ABB RAPID module: ComBase_LU.sys

MODULE ComBase_LU(SYSMODULE,NOSTEPIN)
!**********************************************************************
!* Dieses Module definiert  generellen Ablauf / Kommunikation zur SPS *
!* This module defines the general process / communication with PLC   *
!*                                                                    *
!*                Variablen und Einstellungen fuer die SPS            *
!*                   Variables and settings for PLC                   *
!**********************************************************************
! TypID Nummer fuer alle Applikationen
RECORD TypId
  num TypId_num;
ENDRECORD
!Module Version Number
CONST string st_Version_ComBase:="10.3.6c Test ComBase_LU";
 !Update 13th Apr 2015

! Automatische Einstellung der Sprache / Auto Setting for the language
! Abfrage des FlexPendant / request the FlexPendant
! 1=English, 2=Deutsch, 3=???
PERS num n_Sp:=1;
!
! Merker fuer die Applikationen, wird mit PowerOn neu gelesen / Marker for the applications is read when PowerOn
PERS string st_Appl_Info{30,3}:=[["2","Gripp Ware     ","1 = Actuator, 2 = PP->PLC, 3 = Setup"],["24","INOS Best Fit  ","1 = , 2 = , 3 = Setup"],["","",""],["","",""],["","",""],
	["","",""],["","",""],["","",""],["","",""],["","",""],["","",""],["","",""],["","",""],
	["","",""],["","",""],["","",""],["","",""],["","",""],["","",""],["","",""],["","",""],
	["","",""],["","",""],["","",""],["","",""],["","",""],["","",""],["","",""],["","",""],["","",""]];
VAR string st_Appl_Name:="";
VAR string st_Appl_Key{3}:=["","",""];
PERS num n_ApplMax:=2;
PERS num n_Fk4ApplAktiv:=0;
PERS num n_Fk4ApplNum:=0;
PERS bool b_PwOnEnd:=TRUE;
PERS num n_SMPins{4}:=[5553,0,0,0];
TASK PERS bool b_Start_present{30}:=[TRUE,FALSE,TRUE,TRUE,TRUE,TRUE,TRUE,TRUE,TRUE,TRUE,TRUE,TRUE,TRUE,TRUE,TRUE,
								TRUE,TRUE,TRUE,TRUE,TRUE,TRUE,TRUE,TRUE,TRUE,TRUE,TRUE,TRUE,TRUE,TRUE,TRUE];
PERS bool b_ReStart_present{30}:=[TRUE,FALSE,TRUE,TRUE,TRUE,TRUE,TRUE,TRUE,TRUE,TRUE,TRUE,TRUE,TRUE,TRUE,TRUE,
								  TRUE,TRUE,TRUE,TRUE,TRUE,TRUE,TRUE,TRUE,TRUE,TRUE,TRUE,TRUE,TRUE,TRUE,TRUE];
PERS bool b_Stop_present{30}:=[TRUE,FALSE,TRUE,TRUE,TRUE,TRUE,TRUE,TRUE,TRUE,TRUE,TRUE,TRUE,TRUE,TRUE,TRUE,
							   TRUE,TRUE,TRUE,TRUE,TRUE,TRUE,TRUE,TRUE,TRUE,TRUE,TRUE,TRUE,TRUE,TRUE,TRUE];
PERS bool b_Reset_present{30}:=[TRUE,TRUE,TRUE,TRUE,TRUE,TRUE,TRUE,TRUE,TRUE,TRUE,TRUE,TRUE,TRUE,TRUE,TRUE,
								TRUE,TRUE,TRUE,TRUE,TRUE,TRUE,TRUE,TRUE,TRUE,TRUE,TRUE,TRUE,TRUE,TRUE,TRUE];
PERS bool b_StartUser_present:=TRUE;
PERS bool b_ReStartUser_present:=TRUE;
PERS bool b_StopUser_present:=TRUE;
PERS bool b_ResetUser_present:=TRUE;
PERS bool b_PPMoved:=FALSE;
VAR bool b_PPMoved_mem:=FALSE;

VAR num n_Appl_count;
VAR bool b_UserEv;
!
! Variablen zum Dialog / Varaiables for Dialog
VAR string st_UiHeader{3};
VAR string st_UiHeader_2{3};
VAR string st_UiMsgLines{5};
VAR string st_UiMsgLine1{3};
VAR string st_UiMsgLine2{3};
VAR string st_UiMsgLine3{3};
VAR string st_UiMsgLine4{3};
VAR string st_UiMsgLine5{3};
VAR listitem li_UiMsgList{5};
VAR string st_UiMsgButtons{5};
VAR string st_UiMsgButtons1{3};
VAR string st_UiMsgButtons2{3};
VAR string st_UiMsgButtons3{3};
VAR string st_UiMsgButtons4{3};
VAR string st_UiMsgButtons5{3};
VAR string st_Dummy{3};
VAR string st_Dummy2{3};
VAR btnres br_UiAnswer;
!----------------------------------------------------
!Predefined Const for TypID
!
CONST TypId Id_00:=[0];
CONST TypId Id_01:=[1];
CONST TypId Id_02:=[2];
CONST TypId Id_03:=[3];
CONST TypId Id_04:=[4];
CONST TypId Id_05:=[5];
CONST TypId Id_06:=[6];
CONST TypId Id_07:=[7];
CONST TypId Id_08:=[8];
CONST TypId Id_09:=[9];
CONST TypId Id_10:=[10];
CONST TypId Id_11:=[11];
CONST TypId Id_12:=[12];
CONST TypId Id_13:=[13];
CONST TypId Id_14:=[14];
CONST TypId Id_15:=[15];
!----------------------------------------------------
! Variablen und Einstellungen der MsgBox die von den Appl gemeinsam genutzt werden /
! Variables and settings of the MsgBox that are shared by all Applications
VAR string st_MsgBoxHeader{3};
VAR string st_MsgBoxLine3{3};
VAR string st_MsgBoxLine4{3};
VAR string st_MsgBoxLine5{3};
VAR string st_MsgBoxElogLine4;
VAR string st_MsgBoxbutton1{3};
VAR string st_MsgBoxbutton2{3};
VAR string st_MsgBoxbutton3{3};
VAR string st_MsgBoxbutton4{3};
VAR string st_MsgBoxbutton5{3};
VAR string st_MsgBoxSignal;
VAR string st_MsgBoxSignalValue;
VAR string st_MsgBoxGeraeteName{3};
VAR num n_MsgBoxApplError;
VAR num n_MsgBoxPLC_Error;
VAR num n_MsgBoxGeraeteNr;
VAR num n_MsgBoxAnswer;
VAR num n_Step;
!----------------------------------------------------
! Variablen und Einstellungen der MsgBoxEventStart die von den Appl gemeinsam genutzt werden /
! Variables and settings of the MsgBoxEventStart that are shared by all Applications
VAR string st_MsgBoxEvHeader{3};
VAR string st_MsgBoxEvLine3{3};
VAR string st_MsgBoxEvLine4{3};
VAR string st_MsgBoxEvLine5{3};
VAR string st_MsgBoxEvElogLine4;
VAR string st_MsgBoxEvbutton1{3};
VAR string st_MsgBoxEvbutton2{3};
VAR string st_MsgBoxEvbutton3{3};
VAR string st_MsgBoxEvbutton4{3};
VAR string st_MsgBoxEVbutton5{3};
VAR string st_MsgBoxEvSignal;
VAR string st_MsgBoxEvSignalValue;
VAR string st_MsgBoxEvGeraeteName{3};
VAR num n_MsgBoxEvApplError;
VAR num n_MsgBoxEvPLC_Error;
VAR num n_MsgBoxEvGeraeteNr;
VAR num n_MsgBoxEvAnswer;
VAR num n_StepEv;
!----------------------------------------------------
! Kalibrierposition jpCalibA1_A6 Achsen1-6 auf 0 Grad / Calibration position
CONST jointtarget jpCalibA1_A6:=[ [ 0, 0, 0, 0, 0, 0],[0, 0, 0, 0, 0, 0]];
PERS jointtarget jpTemp:=[ [ 92.8961, 38.0687, 0, 0, 2, 1.67904E-07],[9E+09, 9E+09, 9E+09, 9E+09, 9E+09, 9E+09]];
!
VAR num n_HomeSelect;
VAR num n_PGNNumber;
PERS num n_PGNNumber_Mem:=1;!Last Program number memory

VAR num n_Temp;
VAR bool b_Temp;
VAR num n_JobFinNum;
VAR num n_JobReqNum;
VAR bool b_JobF_w;
VAR bool b_JobR_w;


!----------------------------------------------------
! Tool fuer Position jpSM1SyncSwitch / Tool information for jpSM1SyncSwitchpos position
TASK PERS tooldata t_SMSync:= [TRUE, [[0.04, -0.03, 66.92], [0.991445, 0, 0, 0.130526]],[26.5, [-58.6, 41.7, -18.4],[1, 0, 0, 0], 0, 0, 0.141]];
!
!**********************************************************
!Copy SM Files to HOME directory                         *
!**********************************************************
CONST string stSMCalInternal:="INTERNAL:/OPTIONS/PSC/psc_calib_";
CONST string stSMCalHome:="HOME:/SafetyBCK/psc_calib_";
CONST string stSMInternal:="INTERNAL:/OPTIONS/PSC/psc_user_";
CONST string stSMHome:="HOME:/SafetyBCK/psc_user_";
CONST string stSMBck:="/hd0a/BACKUP/";
CONST string stSMBckFile:="/HOME/SafetyBCK/psc_user_";
CONST string stSMBckCal:="/HOME/SafetyBCK/psc_calib_";

VAR string stCon_Int_Dir;  !Controller internal directory
VAR string stCon_Home_Dir; !Controller internal Home directory
VAR string sthd0a_Home_Dir;!Flash card internal Home directory

! Filesize of an empty SM user_config
CONST num nSMFilesize:=230;
!----------------------------------------------------
! Home Var
TASK PERS tooldata t_Home:= [TRUE, [[26.5774, 98.0613, 502.695], [0.608761, 0, 0, -0.793353]],[311.4, [-15.6, -0.4, 261.4],[1, 0, 0, 0], 130.469, 118.237, 123.004]];
TASK PERS wobjdata wobj_home:=[FALSE, TRUE, "", [[603,2050.01,-515], [0,0,0,1]], [[0,0,0], [1,0,0,0]]];
VAR speeddata sp_SpeedHome;
VAR listitem listHome{5};
!----------------------------------------------------
! Bezeichner fuer die Home, bleibt einsprachig / Identifier for the home, remains monolingual
CONST listitem listHomeConst{5} := [ ["","Home 1 "], ["","Home 2 "],["","Home 3 "],["","Home 4 "] ,["","Home 5 "]  ];
!----------------------------------------------------
! Home Posabweichung Fein 2 Grad fuer Weltzone Home Ueberwachung / Home position in position tolerance
CONST jointtarget delta_HomePosFine := [ [ 2, 2, 2, 2, 2, 2],[5, 5, 5, 5, 5, 5]];
!----------------------------------------------------
! Volumen-Daten Weltzone Home Ueberwachung / Volume of data world-zone Home Surveillance
VAR shapedata sh_HomePos1;
VAR shapedata sh_HomePos2;
VAR shapedata sh_HomePos3;
VAR shapedata sh_HomePos4;
VAR shapedata sh_HomePos5;
!----------------------------------------------------
! Weltzonen Home Ueberwachung / World Home Surveillance Zones
VAR wzstationary wz_HomePos1:=[0];
VAR wzstationary wz_HomePos2:=[0];
VAR wzstationary wz_HomePos3:=[0];
VAR wzstationary wz_HomePos4:=[0];
VAR wzstationary wz_HomePos5:=[0];
!----------------------------------------------------
! Kugel durchmesser Weltzonen Ueberwachung / Ball diameter world zones Surveillance
CONST num n_Ball:=50;
!----------------------------------------------------
! Merker fuer Kolisionsueberwachung / Marker for Collision control
PERS bool b_CollZoneOccupied{63}:=[FALSE,FALSE,FALSE,FALSE,FALSE,FALSE,FALSE,FALSE,FALSE,FALSE,FALSE,FALSE,FALSE,FALSE,FALSE,FALSE,FALSE,FALSE,FALSE,FALSE,FALSE,FALSE,FALSE,FALSE,FALSE,FALSE,FALSE,FALSE,FALSE,FALSE,FALSE,FALSE,FALSE,FALSE,FALSE,FALSE,FALSE,FALSE,FALSE,FALSE,FALSE,FALSE,FALSE,FALSE,FALSE,FALSE,FALSE,FALSE,FALSE,FALSE,FALSE,FALSE,FALSE,FALSE,FALSE,FALSE,FALSE,FALSE,FALSE,FALSE,FALSE,FALSE,FALSE];
PERS num n_Coll{5}:=[2,0,0,0,0];
PERS num n_CollClZ:=1;
PERS bool b_CollClearAct:=FALSE;
!----------------------------------------------------
! Merker fuer PP wurde versetzt
VAR bool b_CheckPP;
!----------------------------------------------------
! Fehlerausgabe Status / Error Status
VAR bool b_OK;
VAR bool b_TimeOut;
!----------------------------------------------------
! Merker fuer Produktions loop / Marker for production loops
VAR bool b_AutoOff;
! Betriebsstundenzaehler / operating hours counters
VAR string st_op_cnt:="";
PERS num n_op_h_counter:=5881;
VAR string st_Abs;
!----------------------------------------------------
VAR Bool b_MainProg_Started ;!A main program as been started
PERS Bool b_PowerOn_exe_OK:=TRUE ;!Power on event has been executed
PERS Bool b_TbCom_Started:=TRUE ;!Background TB Com started
PERS bool b_Ignore_NoAppl_Chk:=FALSE ;!Ignore No APpplication check in StartCOM
PERS num n_ModeOP_Mem:=1 ;!Keyswitch mode operation memory
VAR Bool b_PathColDetectOn:=FALSE ;!Motor supervision on
VAR num n_ManSyncCMD:=0;! ManSyncPos Command
!----------------------------------------------------
!Variables to Check if this robot absolute accuracy compitable
PERS String st_RobotType:="ROB1_7600_2.55_500" ;!Robot type
PERS Bool b_Robot_ABS_Type ;!Robot is absolute accurate
VAR Bool b_ABS_Acc_Enable:=TRUE ;!Application ignore Absolute accuracy message
!----------------------------------------------------

!MsgBox di Break Control
PERS String st_MsgboxBrk_SignalName ;!Message box break Signal name to TB_Com
PERS String st_MsgboxBrk_ReturnName ;!Message box break Return Signal name from TB_Com
PERS Dnum dn_MsgboxBrk_ReqValue ;!Message box break required value to TB_Com
PERS Bool b_Invert_Control ;!Message box break Inverse Control Output to TB_Com

!Variables for monitoring Safety Gate and Manual teach mode keyswitch
PERS Bool b_SafetyGate_Was_Opened ;!Safety Gate was opened
PERS Bool b_ManMode_Was_Selected ;!Manual mode was selected
PERS Num n_SafetyGate_Req_Time;! Time the safety gate must be opened before timeout
PERS Num n_SafetyGate_Opened_Time;! Time the safety gate has been opened

!Variables for Log system
PERS String s_LOG_TX_Data ;!Message to be entered into log max 50 char
PERS String s_LOG_TX_Cat  ;!Message Category into log max 4 char

!Variables for Bit level Group Input and Output control
VAR num  n_LastGroupOutput:=0;
VAR num  n_LastGroupInput:=0;

!Robot number used identify the robot used for this task mainly used for Multimove
CONST Num n_RobotNr:=1;

!Memorise plc Error code
PERS Num n_PLC_ErrCode_Mem:=-4;
!----------------------------------------------------


!Variables for Indirect_WOBJ
PERS num n_DefWob_jDiff_Ges{3}:=[2.09808E-05,0.264905,0.433745];
PERS num n_DefWobj_Diff_Z{3}:=[2.09808E-05,-0.00128365,0.00133324];
PERS num n_DefWobj_Diff_Y{3}:=[0,0.264893,-0.417847];
PERS num n_DefWobj_Diff_X{3}:=[0,-0.0022583,-0.116348];
PERS wobjdata wobj_DefWobj_car0:=[FALSE,TRUE,"",[[-1.55826,939.221,447.268],[0.707962,0.0617476,0.0581078,-0.701142]],[[0,0,0],[1,0,0,0]]];
PERS tooldata t_DefWobj_Act_tool:=[TRUE,[[0,0,0],[1,0,0,0]],[0.001,[0,0,0.001],[1,0,0,0],0,0,0]];
PERS wobjdata wobj_DefWobj_ACT_wobj:=[FALSE,TRUE,"",[[0,0,0],[1,0,0,0]],[[0,0,0],[1,0,0,0]]];
PERS string s_DefWobj_Tool_Name:="tool0";
PERS string s_DefWobj_Wobj_Name:="wobj0";
PERS num n_DefWobj_px:=2734.52;
PERS num n_DefWobj_py:=-250;
PERS num n_DefWobj_pz:=40.459;
PERS robtarget rt_DefWobj_user_p{3}:=[[[271.15,-1260.46,24.4443],[0.539391,-0.00995541,0.0179942,0.841804],[-1,-1,0,1],[9E+09,9E+09,9E+09,9E+09,9E+09,9E+09]],[[275.724,-1760.69,26.8719],[0.539275,-0.00995293,0.0180075,0.841877],[-1,-1,0,1],[9E+09,9E+09,9E+09,9E+09,9E+09,9E+09]],[[-224.132,-1764.6,23.8962],[0.539218,-0.00994843,0.0180428,0.841914],[-2,-2,0,1],[9E+09,9E+09,9E+09,9E+09,9E+09,9E+09]]];
PERS robtarget rt_DefWobj_mess_p{3}:=[[[2242.11,250,-46.365],[1,0,0,0],[-1,-1,-1,0],[9E+09,9E+09,9E+09,9E+09,9E+09,9E+09]],[[2734.52,250,40.459],[1,0,0,0],[-1,-1,-1,0],[9E+09,9E+09,9E+09,9E+09,9E+09,9E+09]],[[2734.52,-250,40.459],[1,0,0,0],[-1,-1,-1,0],[9E+09,9E+09,9E+09,9E+09,9E+09,9E+09]]];


!----------------------------------------------------

PROC InitAutoMode()
!******************************************************
!*                                                    *
!* Prozedur fuer das Starten des Roboters in Automatik*
!*   Procedure for starting the robot in automatic!   *
!*                                                    *
!******************************************************
!
! Bewegungsueberwachung einschalten / Activate motion supervision
MotionSup \On;

!Reset Msgbox signals
SetGO PLC_go_ErrCode, 0;
Reset PLC_do_MsgToPLC;
Reset PLC_do_ErrorToPLC;
Reset PLC_do_StopToPLC;
Reset VB_do_TaskBrake;
n_PLC_ErrCode_Mem:=-1;

! abfrage ob Betriebsart Hand / Check operation mode
WHILE OpMode()= OP_AUTO DO
	st_UiHeader:=["Com, Waiting for Robot in Teach Mode ","Com, Warte auf Hand-Betrieb","???"];
	st_UiMsgLine1:=["  Please switch the mode selection ","  Bitte Programm Main in der Betriebsart ","???"];
	st_UiMsgLine2:=["  to Teach/Manual Mode.","  Hand starten.","???"];
	UIMsgBox\Header:=st_UiHeader{n_Sp},st_UiMsgLine1{n_Sp}\MsgLine2:=st_UiMsgLine2{n_Sp}
	\Buttons:=btnOK\Icon:=iconWarning;
	!
	IF OpMode()= OP_AUTO Stop;
ENDWHILE

IF b_PowerOn_exe_OK=FALSE PowerOnCom ;

! Abfrage ob die AbsAcc ein ist
ReadCfgData "/MOC/ROBOT/ROB_1","use_robot_calib",st_Abs;

IF st_Abs="r1_uncalib" AND b_Robot_ABS_Type THEN
	st_UiHeader:=["Com, No Absolute Accuracy","Com, Keine Absolutgenauigkeit","???"];
	st_UiMsgLine1:=["Warning! The robot absolute accuracy is turned Off.","Achtung bei diesem Roboter ist die Absolutgenauigkeit = Off","???"];
	st_UiMsgLine2:=["Absolute accuracy must be enabled","Ohne aktive Absolutgenauigkeit ist es nicht erlaubt","???"];
	st_UiMsgLine3:=["and without it, there is a high risk ","den Roboter zu programmieren oder Programme abzufahren,","???"];
	st_UiMsgLine4:=["of a collision.","es besteht Kollisionsgefahr!","???"];
	st_UiMsgLine5:=["Please ensure it is enabled!","Bitte schalten Sie die Absolutgenauigkeit wieder ein!","???"];
    st_UiMsgButtons5:=["Ignore","ignorieren","???"];
    st_UiMsgButtons:=["","","","",st_UiMsgButtons5{n_Sp}];
    st_UiMsgLines:=[st_UiMsgLine1{n_Sp},st_UiMsgLine2{n_Sp},st_UiMsgLine3{n_Sp},st_UiMsgLine4{n_Sp},st_UiMsgLine5{n_Sp}];
    br_UiAnswer:=UIMessageBox (\Header:=st_UiHeader{n_Sp}\MsgArray:=st_UiMsgLines\BtnArray:=st_UiMsgButtons\Icon:=iconError);
ENDIF

! Abfrage ob der Roboter synchron ist / check because synced Robot
IF DOutput(SM1_do_Synced) = 0 THEN
	br_UiAnswer:=0;
	st_UiHeader:=["Com, SafeMove not Synchronised!","Com, SafeMove nicht synchron!","???"];
	st_UiMsgLine1:=["Warning! SafeMove(safety control) is not activated","Achtung, SafeMove(Sicherheitssteuerung) ist nicht aktiv!","???"];
	st_UiMsgLine2:=["Automatic operation without *SoftSync* is not possible!","Automatikbetrieb ist mit der Option *SoftSync* nicht moeglich!","???"];
	st_UiMsgLine3:=["Please synchronise the robot (SafeMove).","Bitte den Roboter (SafeMove) erst manuell synchronisieren lassen.","???"];
	st_UiMsgLine4:=["","","???"];
	st_UiMsgLine5:=["Press> Ignore to continue to operate without SoftSync.","Mit ignorieren geht es im Ablauf (ohne SoftSync) weiter.","???"];
	st_UiMsgButtons5:=["Ignore","ignorieren","???"];
	st_UiMsgButtons:=["","","","",st_UiMsgButtons5{n_Sp}];
	st_UiMsgLines:=[st_UiMsgLine1{n_Sp},st_UiMsgLine2{n_Sp},st_UiMsgLine3{n_Sp},st_UiMsgLine4{n_Sp},st_UiMsgLine5{n_Sp}];
	!
	br_UiAnswer:=UIMessageBox (\Header:=st_UiHeader{n_Sp}
	\MsgArray:=st_UiMsgLines\BtnArray:=st_UiMsgButtons\Icon:=iconWarning);
ENDIF

! Simulierte Signale Abfragen
IF DOutput(VB_do_Simulated_IO)= 1 AND RobOS() = TRUE  THEN
	WHILE DOutput(VB_do_Simulated_IO)= 1 DO
 		st_UiHeader:=["Com, Caution simulated signals!","Com, Achtung Simulierte Signale!","???"];
 		st_UiMsgLine1:=["There are some signals that are simulated which is not allowed in ","Das Simulieren von Signalen ist im Automatik nicht erlaubt!","???"];
 		st_UiMsgLine2:=["automatic mode!  To continue please","Um fortzufahren bitte die Simulation aller","???"];
 		st_UiMsgLine3:=["select the I/O menu then turn off the simulation/s.","Signale im Ein-Ausgangs Fenster ausschalten.","???"];
 		UIMsgBox\Header:=st_UiHeader{n_Sp},st_UiMsgLine1{n_Sp}\MsgLine2:=st_UiMsgLine2{n_Sp}\MsgLine3:=st_UiMsgLine3{n_Sp}
 						\Buttons:=btnOk\Icon:=iconWarning;
		!
		IF DOutput(VB_do_Simulated_IO)= 1 Stop;
	ENDWHILE
ENDIF

!Jog supervision enable
WriteCfgData "/MOC/MOTION_SUP/rob1","jog_col_detect_on", TRUE;

!Check motor supervision enabled
ReadCfgData "/MOC/MOTION_SUP/rob1","path_col_detect_on",b_PathColDetectOn;

IF b_PathColDetectOn=FALSE THEN
	st_UiHeader:=["Com, Motor Supervision","Com, Motor Ueberwachung","???"];
	st_UiMsgLine1:=["The robot path supervision is","Die Roboter Pfad Ueberwachung ist","???"];
	st_UiMsgLine2:=["turned off and should be turned on.","ausgeschalten und solle angeschalten sein.","???"];
	st_UiMsgLine3:=["","","???"];
	st_UiMsgLine4:=["","","???"];
	st_UiMsgLine5:=["Please select option.","Option waehlen bitte.","???"];
    st_UiMsgButtons4:=["Turn On","anschalten","???"];
    st_UiMsgButtons5:=["Ignore","ignorieren","???"];
    st_UiMsgButtons:=["","","",st_UiMsgButtons4{n_Sp},st_UiMsgButtons5{n_Sp}];
    st_UiMsgLines:=[st_UiMsgLine1{n_Sp},st_UiMsgLine2{n_Sp},st_UiMsgLine3{n_Sp},st_UiMsgLine4{n_Sp},st_UiMsgLine5{n_Sp}];
    br_UiAnswer:=UIMessageBox (\Header:=st_UiHeader{n_Sp}\MsgArray:=st_UiMsgLines\BtnArray:=st_UiMsgButtons\Icon:=iconWarning);

    IF br_UiAnswer=4 WriteCfgData "/MOC/MOTION_SUP/rob1","path_col_detect_on", TRUE;
ENDIF

! meldet an PLC das Programmzeiger im Main ist / Inform PLC main program is selected
b_CheckPP:=TRUE;
Set SYS_do_MainStarted;
VelSet 100,5000;

! zum anfahren der Homeposition
! abfrage ob mehr als eine HomePos / Check number of homes configured
FOR i FROM 1 TO 5 DO
  IF b_HomeInUse{i}=TRUE Incr n_Temp;
ENDFOR

! auslesen der Beschreibung der benutzten Home / Read the home descriptions
IF n_Temp>1 THEN
 	Abfrg2:
	FOR i FROM 1 TO 5 DO
		IF b_HomeInUse{i} THEN
			! vorgabe der Home von der SPS / specification of the Home of the PLC
			IF b_PLCNeedHome(i)= TRUE THEN
				st_UiMsgLine1:=["PLC> ","SPS> ","???"];
				listHome{i}.text:=st_UiMsgLine1{n_Sp};
			ELSE
				listHome{i}.text:="        ";
			ENDIF
			listHome{i}.text:=listHome{i}.text+listHomeConst{i}.text+st_Home_label{i};
		ELSE
			listHome{i}.text:="";
		ENDIF
	ENDFOR

	! Anzeigen der HomePos / Generate Home positions message
  	st_UiHeader:=["Com, The Robot is ","Com, Der Roboter steht auf ","???"];

	IF n_RobInHomeDO()> 0 THEN
    	st_UiHeader_2:=["at Home number "+ValToStr(n_RobInHomeDO()),"Home "+ValToStr(n_RobInHomeDO()),"???"+ValToStr(n_RobInHomeDO())];
	ELSE
    	st_UiHeader_2:=["not in any Home.","keiner Home.","???"];
	ENDIF

	st_UiMsgButtons1:=["Refresh Display","Ansicht aktualisieren","???"];
	st_UiMsgButtons4:=["Ok","Ok","???"];
	st_UiMsgButtons5:=["Abort","Abbruch","???"];
	st_UiMsgButtons:=[st_UiMsgButtons1{n_Sp},"","",st_UiMsgButtons4{n_Sp},""];

	n_HomeSelect := UIListView(\Result:=br_UiAnswer\Header:=st_UiHeader{n_Sp}+st_UiHeader_2{n_Sp},listHome
      \BtnArray:=st_UiMsgButtons\Icon:=iconInfo\DefaultIndex:=n_RobInHomeDO());

	IF br_UiAnswer = 1 GOTO Abfrg2;
	IF br_UiAnswer = 5 THEN
  	TPErase;
  	TPShow TP_LATEST;
  	EXIT ;
   ENDIF
ELSE !n_temp>1
	! es gibt nur eine Home / There is only one Home
	n_HomeSelect:=1;
ENDIF !n_temp>1

!----------------------------------------------------
! Ueberprueft ob die Homeposition programmiert wurde / Checks whether the home position has been programmed
br_UiAnswer:=0;
b_Temp:=FALSE;
IF n_HomeSelect=1 AND jpHome1.robax <> jpCalibA1_A6.robax AND b_HomeAkt{n_HomeSelect}=TRUE b_Temp:=TRUE;
IF n_HomeSelect=2 AND jpHome2.robax <> jpCalibA1_A6.robax AND b_HomeAkt{n_HomeSelect}=TRUE b_Temp:=TRUE;
IF n_HomeSelect=3 AND jpHome3.robax <> jpCalibA1_A6.robax AND b_HomeAkt{n_HomeSelect}=TRUE b_Temp:=TRUE;
IF n_HomeSelect=4 AND jpHome4.robax <> jpCalibA1_A6.robax AND b_HomeAkt{n_HomeSelect}=TRUE b_Temp:=TRUE;
IF n_HomeSelect=5 AND jpHome5.robax <> jpCalibA1_A6.robax AND b_HomeAkt{n_HomeSelect}=TRUE b_Temp:=TRUE;

IF b_Temp=FALSE THEN
	st_UiHeader:=["Com, Home Configuration Error","Com, Fehlerhafte Home_","Com,???"];
	IF b_HomeAkt{n_HomeSelect}=FALSE THEN
		st_UiMsgLine1:=["The Home position selected has not been activated","Die ausgewaehlte Home ist nicht aktiv","???"];
		st_UiMsgLine2:=["therefore, the Home output will not be sent to the PLC.","der Ausgang wird nicht zur SPS gesetzt.","???"];
		st_UiMsgLine3:=["Please select 'HomeSetup' to configure.","Bitte ueber das HomeSetup die Home aktivieren.","???"];
	ELSE
		st_UiMsgLine1:=["The Home position selected either not programmed","Die ausgewaehlte Home ist nicht programmiert","???"];
		st_UiMsgLine2:=["or the robot is in the calibration position!","oder entspricht der Nullstellung!","???"];
		st_UiMsgLine3:=["Please select 'Setup' to configure.","Bitte die Position ueber das HomeSetup anpassen.","???"];
	ENDIF

	st_UiMsgButtons3:=["Home Setup","Home Setup","???"];
	st_UiMsgButtons5:=["Abort","Abbruch","???"];
	st_UiMsgButtons:=["","",st_UiMsgButtons3{n_Sp},"",st_UiMsgButtons5{n_Sp}];
	st_UiMsgLines:=[st_UiMsgLine1{n_Sp},st_UiMsgLine2{n_Sp},st_UiMsgLine3{n_Sp},"",""];

	br_UiAnswer:=UIMessageBox (\Header:=st_UiHeader{n_Sp}+ValToStr(n_HomeSelect)
		\MsgArray:=st_UiMsgLines\BtnArray:=st_UiMsgButtons\Icon:=iconWarning);

	IF br_UiAnswer = 5 THEN
		TPErase;
		TPShow TP_LATEST;
		EXIT;
	ENDIF

	IF br_UiAnswer = 3 Homesetup;
	EXIT;
ENDIF

! Abfrage wegen Tool 0 / check because of tool zero
IF CTool()=tool0 THEN
  	br_UiAnswer:=0;
  	st_UiHeader:=["Com, Tool Load check","Com, Tool Ueberpruefung","???"];
  	st_UiMsgLine1:=["Attention!! the active tool is tool0.","Achtung das aktive Tool ist - tool0 - !!! ","???"];
  	st_UiMsgLine2:=["The robot cannot move with tool0 because","Der Roboter kann vermutlicht wegen falschen  ","???"];
  	st_UiMsgLine3:=["it has the incorrect payload configured.","Gewichtsdaten nicht bewegt werden, ","???"];
  	st_UiMsgLine4:=["Using the Jogging Window, please change to the","bitte waehle im Bewegen-Fenster das richtige Tool aus,","???"];
  	st_UiMsgLine5:=["correct tool then select 'Ok' button.","bevor es mit Ok weiter geht.","???"];
  	st_UiMsgButtons1:=["","","???"];
  	st_UiMsgButtons2:=["","","???"];
  	st_UiMsgButtons3:=["","","???"];
  	st_UiMsgButtons4:=["Ok","Ok","???"];
  	st_UiMsgButtons5:=["","","???"];
  	st_UiMsgButtons:=[st_UiMsgButtons1{n_Sp},st_UiMsgButtons2{n_Sp},st_UiMsgButtons3{n_Sp},st_UiMsgButtons4{n_Sp},st_UiMsgButtons5{n_Sp}];
  	st_UiMsgLines:=[st_UiMsgLine1{n_Sp},st_UiMsgLine2{n_Sp},st_UiMsgLine3{n_Sp},st_UiMsgLine4{n_Sp},st_UiMsgLine5{n_Sp}];
  	!
  	br_UiAnswer:=UIMessageBox (\Header:=st_UiHeader{n_Sp}
  	\MsgArray:=st_UiMsgLines\BtnArray:=st_UiMsgButtons\Icon:=iconWarning);
ENDIF

! Bestaetigung und Geschwindigkeitsauswahl / Confirmation and speed selection
sp_SpeedHome:=v100;
IF b_RobInHomeDO(n_HomeSelect)= FALSE THEN
  	br_UiAnswer:=0;
  	st_UiHeader:=["Com, Move Robot to Homepos ","Com, Bewege Roboter zur Home ","Com,???"];
  	st_UiMsgLine3:=["     Attention!","    Achtung!","???"];
  	st_UiMsgLine4:=["     The Robot will move -> ","    Roboter faehrt mit Ok -> ","???"];
  	st_UiMsgLine5:=["     directly to the Home ","    direkt zur Home ","???"];
  	st_UiMsgButtons1:=["Fast (v250)","SCHNELL (v250)","???"];
  	st_UiMsgButtons2:=["Slow (v100)","LANGSAM (v100)","???"];
  	st_UiMsgButtons3:=["","","???"];
  	st_UiMsgButtons4:=["Move Home","Ok","???"];
  	st_UiMsgButtons5:=["Abort","Abbruch","???"];
  	st_UiMsgButtons:=[st_UiMsgButtons1{n_Sp},st_UiMsgButtons2{n_Sp},st_UiMsgButtons3{n_Sp},st_UiMsgButtons4{n_Sp},""];
  	st_Dummy:=st_UiMsgButtons2;
  	Abfrg1:
  	st_UiMsgLines:=[" "," ",st_UiMsgLine3{n_Sp},st_UiMsgLine4{n_Sp}+st_Dummy{n_Sp},st_UiMsgLine5{n_Sp}+ValToStr(n_HomeSelect)];

  	br_UiAnswer:=UIMessageBox (\Header:=st_UiHeader{n_Sp}+ValToStr(n_HomeSelect)
  			\MsgArray:=st_UiMsgLines\BtnArray:=st_UiMsgButtons\Icon:=iconWarning);

	TEST br_UiAnswer
		CASE 1:
		! schnell/fAST
		st_Dummy:=st_UiMsgButtons1;
		sp_SpeedHome:=v200;
		GOTO Abfrg1;
	CASE 2:
		! langsam/sLOW
		st_Dummy:=st_UiMsgButtons2;
		sp_SpeedHome:=v100;
		GOTO Abfrg1;
	CASE 4:
		! OK/ok
	CASE 5:
		! Abbruch / Abort
		TPErase;
		TPShow TP_LATEST;
			EXIT;
	ENDTEST

	! Prozedur zum Initialisieren von Ein-, Ausgaengen, Variabelen fuer den User / Procedure to initialize inputs, outputs, variables for the user
	InitBeforHome n_HomeSelect;
	! Homefahrt
	t_Home := CTool();
	wobj_home := CWobj();

	TEST n_HomeSelect
	CASE 1:
		MoveAbsJ jpHome1\NoEOffs, sp_SpeedHome, fine, t_Home\WObj:=wobj_home;
	CASE 2:
		MoveAbsJ jpHome2\NoEOffs, sp_SpeedHome, fine, t_Home\WObj:=wobj_home;
	CASE 3:
		MoveAbsJ jpHome3\NoEOffs, sp_SpeedHome, fine, t_Home\WObj:=wobj_home;
	CASE 4:
		MoveAbsJ jpHome4\NoEOffs, sp_SpeedHome, fine, t_Home\WObj:=wobj_home;
	CASE 5:
		MoveAbsJ jpHome5\NoEOffs, sp_SpeedHome, fine, t_Home\WObj:=wobj_home;
	ENDTEST
ELSE !n_HomeSelect
	! Roboter steht schon auf Home x
	! Prozedur zum Initialisieren von Ein-, Ausgaengen, Variabelen fuer den User /
	! Robots already standing at home x
	! Procedure to initialize inputs, outputs, variables for the user
 	InitBeforHome n_HomeSelect;
ENDIF !n_HomeSelect

! check ob Home x Ausgang = 1
IF b_RobInHomeDO(n_HomeSelect)= FALSE THEN
  	br_UiAnswer:=0;
  	st_UiHeader:=["Com, Error Output SYS_do_Home_"+ValToStr(n_HomeSelect)+" = 0","Com, Fehler: Ausgang SYS_do_Home_"+ValToStr(n_HomeSelect)+" = 0","Com,???"];
  	st_UiMsgLine3:=[" Attention Output from Home "+ValToStr(n_HomeSelect)+" does not =1.","Achtung der Ausgang fuer die Home " +ValToStr(n_HomeSelect)+" wurde nicht gesetzt!","???"];
  	st_UiMsgLine4:=[" The HomePos is not valid therefore, the program will stop.","Die Grundstellung ist nicht gueltig, der Ablauf wird abgebrochen.","???"];
  	st_UiMsgLine5:=[" Please ReCheck the Home"+ValToStr(n_HomeSelect)+" using the HomeSetup option.","Bitte im HomeSetup die Grundstellung Home"+ValToStr(n_HomeSelect)+"  berichtigen. ","???"];
  	st_UiMsgButtons1:=["","","???"];
  	st_UiMsgButtons2:=["","","???"];
  	st_UiMsgButtons3:=["Home Setup","Home Setup","???"];
  	st_UiMsgButtons4:=["Ok","Ok","???"];
  	st_UiMsgButtons5:=["","","???"];
  	st_UiMsgButtons:=[st_UiMsgButtons1{n_Sp},st_UiMsgButtons2{n_Sp},st_UiMsgButtons3{n_Sp},st_UiMsgButtons4{n_Sp},st_UiMsgButtons5{n_Sp}];
  	st_UiMsgLines:=[" "," ",st_UiMsgLine3{n_Sp},st_UiMsgLine4{n_Sp},st_UiMsgLine5{n_Sp}];
  	!
  	br_UiAnswer:=UIMessageBox (\Header:=st_UiHeader{n_Sp}\MsgArray:=st_UiMsgLines\BtnArray:=st_UiMsgButtons\Icon:=iconError);
  	! Fehler /Error
    IF br_UiAnswer = 3 Homesetup;
  	TPErase;
  	TPShow TP_LATEST;
 	EXIT;
ENDIF

InitInHome n_HomeSelect;

! Prozedur zum Initialisieren von Ein-, Ausgaengen, Variabelen fuer den User /
! Procedure to initialize user inputs, outputs and variables
InitMain;
InitProduktion;

WHILE OpMode()<>OP_AUTO DO
	! Aufforderung fuer Automaikbetrieb
	br_UiAnswer:=0;
	st_UiHeader:=["Com, Automatic Mode","Com, Automatik Extern Betrieb","Com,???"];
	st_UiMsgLine2:=["Please turn the mode selection Switch ","Den Schluesselschalter auf Automatik stellen ","???"];
	st_UiMsgLine3:=["to the Automatic Mode External position.","um in die Betriebsart Automatik Extern ","???"];
	st_UiMsgLine4:=[" ","zu wechseln.","???"];
	st_UiMsgButtons5:=["Abort","Abbruch","???"];
	st_UiMsgButtons:=["","","","",""];
	st_UiMsgLines:=[" ",st_UiMsgLine2{n_Sp},st_UiMsgLine3{n_Sp},st_UiMsgLine4{n_Sp},""];

	br_UiAnswer:=UIMessageBox (\Header:=st_UiHeader{n_Sp}
		\MsgArray:=st_UiMsgLines\BtnArray:=st_UiMsgButtons\Icon:=iconInfo\DOBreak:=SYS_do_Auto);
	!
	IF br_UiAnswer = resCancel THEN
		TPErase;
		TPShow TP_LATEST;
		EXIT;
	ENDIF
ENDWHILE

! Schleife fuer den AutoEX Betrieb\Loop for the operational AutoEX
WHILE b_AutoOff=FALSE DO
	b_AutoOff:=FALSE;
	InitProduktion;
	! Betriebsstundenzaehler lesen / operating hours counters read
	st_op_cnt:=GetServiceInfo(ROB_ID \DutyTimeCnt);
	b_Temp:=StrToVal(st_op_cnt, n_op_h_counter);

	WHILE SYS_di_ProgNumValid=1 DO
		st_MsgBoxHeader:=["Com, Error Prog Number Valid ","Com, Fehler Signal Prognum. gueltig!","???"];
		st_MsgBoxLine4:=["The Error is in the PLC","Fehlerbehebung an der SPS","???"];
		st_MsgBoxbutton4:=["Ok","Ok","???"];
		st_MsgBoxSignal:="SYS_di_ProgNumValid";
		st_MsgBoxGeraeteName:=["PLC I/O","SPS E/A","???"];
		n_MsgBoxGeraeteNr:=0;
		st_MsgBoxSignalValue:="0";
		n_MsgBoxApplError:=3;
		n_MsgBoxPLC_Error:=33;
		st_MsgBoxElogLine4:="ComBase/InitAutoMode";
		MsgBox\diBreakSignal:=SYS_di_ErrReset\ErrorToPLC;
	ENDWHILE

	! Betriebsstundenzaehler setzen zur SPS/ operating hours counters set to PLC
	IF b_Temp = TRUE SetGO PLC_go_WeldPoint_Num, n_op_h_counter;
	! anfrage Prognum. / Send program number request
	Set SYS_do_ProgNumReq;

	IF RobOS()  THEN
		st_UiHeader:=["          Com, Program Number","Com, Warte auf gueltige Programmnummer...","Com,???"];
		st_UiMsgLine1:=["         ******************************************","        ******************************************","???"];
		st_UiMsgLine2:=["         *     Waiting for the Program Number     *","        *      Warten auf die Programmnummer     *","???"];
		st_UiMsgLine3:=["         *              from the PLC.         V3.6*","        *               von der SPS.         V3.6*","???"];
		st_UiMsgLine4:=["         ******************************************","        ******************************************","???"];
		! Meldung an SPS, warte auf programmnummer / Waiting PLC Number
		 Reset PLC_do_ErrorToPLC;
		SetGO PLC_go_ErrCode, 32;
		Set PLC_do_MsgToPLC;
  		UIMsgBox\Header:=st_UiHeader{n_Sp},st_UiMsgLine1{n_Sp}\MsgLine2:=st_UiMsgLine2{n_Sp}
				\MsgLine3:=st_UiMsgLine3{n_Sp}\MsgLine4:=st_UiMsgLine4{n_Sp}\Buttons:=btnNone\Icon:=iconInfo
				\DIBreak:=SYS_di_ProgNumValid;
		! zuweisung der Prognum / Allocation of program number
		n_PGNNumber:=GInput(SYS_gi_ProgNumber);
		SetGO PLC_go_ErrCode, 0;
 		Reset PLC_do_MsgToPLC;
 		Reset PLC_do_ErrorToPLC;
	ELSE
		! manuelle Prognr nur fuer RobotStudio / Manual PGNR robot studio
  		st_UiHeader:=[" VirtualProgram Number","Programmnummer Virtual","???"];
 		st_UiMsgLine1:=["Program Number?","Programmnummer? 1-63","???"];
		n_PGNNumber := UINumEntry(\Header:=st_UiHeader{n_Sp}\Message:=st_UiMsgLine1{n_Sp}\Icon:=iconInfo
		\InitValue:=1\MinValue:=1\MaxValue:=63\AsInteger);
	ENDIF
	! Abfrage ob die AbsAcc ein ist
	ReadCfgData "/MOC/ROBOT/ROB_1","use_robot_calib",st_Abs;

	IF st_Abs="r1_uncalib" AND b_Robot_ABS_Type THEN
		st_UiHeader:=["Com, AbsAcc error","Com, Fehler Absolutgenauigkeit","???"];
		st_UiMsgLine1:=["Warning! The robot absolute accuracy is turned Off.","Achtung bei diesem Roboter ist die AbsAcc = Off","???"];
		st_UiMsgLine2:=["Absolute accuracy must be enabled","Ohne aktive Absolutgenauigkeit ist es nicht erlaubt","???"];
		st_UiMsgLine3:=["and without it, there is a high risk","den Roboter zu programmieren oder Programme abzufahren","???"];
		st_UiMsgLine4:=["of a collision.","es besteht Kollisionsgefahr!","???"];
		st_UiMsgLine5:=["Please ensure it is enabled!","Bitte schalten Sie die Absolutgenauigkeit wieder ein!","???"];
		UIMsgBox\Header:=st_UiHeader{n_Sp}, st_UiMsgLine1{n_Sp}\MsgLine2:=st_UiMsgLine2{n_Sp}\MsgLine3:=st_UiMsgLine3{n_Sp}
						\MsgLine4:=st_UiMsgLine4{n_Sp}\MsgLine5:=st_UiMsgLine5{n_Sp}\Buttons:=btnOK\Icon:=iconWarning;
	ENDIF

	n_PGNNumber_Mem:=n_PGNNumber;

	Reset SYS_do_ProgNumReq;
	SetGO PLC_go_WeldPoint_Num,0;
	! aufruf des Programms / Call program number
	Set SYS_do_ApplRun;
	%"Program_"+NumToStr(n_PGNNumber,0)%;
	Reset SYS_do_ApplRun;
ENDWHILE

ERROR
!** Error Handler**
! Fehlerbehandlung von nicht vorhandenen ProgNr. / None existant program number
SkipWarn;
IF ERRNO = ERR_REFUNKPRC THEN
    st_MsgBoxHeader:=["Com, Incorrect Program Number Call ","Com, Falsche Programm Nr. von der SPS!","???"];
    st_Dummy:=["The Routine called Program_"+ValToStr (n_PGNNumber),"Keine Routine Program_"+ValToStr (n_PGNNumber),"???"];
    st_Dummy2:=["was requested but is not programmed!!","im System vorhanden !","???"];
    st_MsgBoxbutton4:=["OK","Ok","???"];
    n_MsgBoxApplError:=0;
    n_MsgBoxPLC_Error:=31;
    st_MsgBoxElogLine4:="ComBase/InitAutoMode";
    MsgBox\diBreakSignal:=SYS_di_ErrReset\Line1:=st_Dummy{n_Sp}\Line2:=st_Dummy2{n_Sp}\ErrorToPLC;
  	TRYNEXT;
ENDIF
SkipWarn;
IF ERRNO = ERR_TP_DOBREAK TRYNEXT;
IF ERRNO = ERR_TP_DIBREAK TRYNEXT;
ENDPROC !(InitAutoMode)

!*******************************************************************************

PROC InitMain()
!**********************
!* Procedure InitMain *
!*   Intialise Main   *
!**********************
! Prozedur zum Initialisieren von Ein-, Ausgaengen, Variabelen / Procedure to initialize inputs, outputs, variables
! Procedur wird 1x im Main aufgerufen / First procedure called from main
 VAR bool b_ComDummy:=FALSE;
 VAR num n_ComDummy:=0;
!
 Reset SYS_do_ProgNumReq;
 Reset SYS_do_ApplRun;
 SetGO PLC_go_ErrCode, 0;
 Reset PLC_do_MsgToPLC;
 Reset PLC_do_ErrorToPLC;
 Reset PLC_do_StopToPLC;
 Reset PLC_do_CollZoneClear;
 Reset PLC_do_CollZoneReq;
 SetGO PLC_go_CollZone, 0;

 CollSafetyInit;
 b_AutoOff:=FALSE;
 n_JobReqNum:=0;
 n_JobFinNum:=0;
 b_JobF_w:=FALSE;
 b_JobR_w:=FALSE;
 !
 Reset PLC_do_Job01_Ready;
 Reset PLC_do_Job02_Ready;
 Reset PLC_do_Job03_Ready;
 Reset PLC_do_Job04_Ready;
 Reset PLC_do_Job05_Ready;
 Reset PLC_do_Job06_Ready;
 Reset PLC_do_Job07_Ready;
 Reset PLC_do_Job08_Ready;
 Reset PLC_do_Job09_Ready;
 Reset PLC_do_Job10_Ready;
 Reset PLC_do_Job11_Ready;
 Reset PLC_do_Job12_Ready;
 Reset PLC_do_Job13_Ready;
 Reset PLC_do_Job14_Ready;
 Reset PLC_do_Job15_Ready;
 Reset PLC_do_Job16_Ready;
 Reset PLC_do_Job17_Ready;
 Reset PLC_do_Job18_Ready;
 Reset PLC_do_Job19_Ready;
 Reset PLC_do_Job20_Ready;
 Reset PLC_do_Job21_Ready;
 Reset PLC_do_Job22_Ready;
 Reset PLC_do_Job23_Ready;
 Reset PLC_do_Job24_Ready;
 Reset PLC_do_Job25_Ready;
 Reset PLC_do_Job26_Ready;
 Reset PLC_do_Job27_Ready;
 Reset PLC_do_Job28_Ready;
 Reset PLC_do_Job29_Ready;
 Reset PLC_do_Job30_Ready;
 Reset PLC_do_Job31_Ready;
 Reset PLC_do_Job32_Ready;
 !
 Reset PLC_do_Job01_Started;
 Reset PLC_do_Job02_Started;
 Reset PLC_do_Job03_Started;
 Reset PLC_do_Job04_Started;
 Reset PLC_do_Job05_Started;
 Reset PLC_do_Job06_Started;
 Reset PLC_do_Job07_Started;
 Reset PLC_do_Job08_Started;
 Reset PLC_do_Job09_Started;
 Reset PLC_do_Job10_Started;
 Reset PLC_do_Job11_Started;
 Reset PLC_do_Job12_Started;
 Reset PLC_do_Job13_Started;
 Reset PLC_do_Job14_Started;
 Reset PLC_do_Job15_Started;
 Reset PLC_do_Job16_Started;
 Reset PLC_do_Job17_Started;
 Reset PLC_do_Job18_Started;
 Reset PLC_do_Job19_Started;
 Reset PLC_do_Job20_Started;
 Reset PLC_do_Job21_Started;
 Reset PLC_do_Job22_Started;
 Reset PLC_do_Job23_Started;
 Reset PLC_do_Job24_Started;
 Reset PLC_do_Job25_Started;
 Reset PLC_do_Job26_Started;
 Reset PLC_do_Job27_Started;
 Reset PLC_do_Job28_Started;
 Reset PLC_do_Job29_Started;
 Reset PLC_do_Job30_Started;
 Reset PLC_do_Job31_Started;
 Reset PLC_do_Job32_Started;
 !
 Reset PLC_do_Typbit_01;
 Reset PLC_do_Typbit_02;
 Reset PLC_do_Typbit_03;
 Reset PLC_do_Typbit_04;
 Reset PLC_do_Typbit_05;
 Reset PLC_do_Typbit_06;
 Reset PLC_do_Typbit_07;
 Reset PLC_do_Typbit_08;
 Reset PLC_do_Typbit_09;
 Reset PLC_do_Typbit_10;
 Reset PLC_do_Typbit_11;
 Reset PLC_do_Typbit_12;
 Reset PLC_do_Typbit_13;
 Reset PLC_do_Typbit_14;
 Reset PLC_do_Typbit_15;
 Reset PLC_do_Typbit_16;
 Reset PLC_do_Typbit_17;
 Reset PLC_do_Typbit_18;
 Reset PLC_do_Typbit_19;
 Reset PLC_do_Typbit_20;
 Reset PLC_do_Typbit_21;
 Reset PLC_do_Typbit_22;
 Reset PLC_do_Typbit_23;
 Reset PLC_do_Typbit_24;
 Reset PLC_do_Typbit_25;
 Reset PLC_do_Typbit_26;
 Reset PLC_do_Typbit_27;
 Reset PLC_do_Typbit_28;
 Reset PLC_do_Typbit_29;
 Reset PLC_do_Typbit_30;
 Reset PLC_do_Typbit_31;
 Reset PLC_do_Typbit_32;

 Reset PLC_do_ServicePos;
 Reset PLC_do_Process_Complete;
 Reset PLC_do_WeldCount;

 !Set output as this robot does not use this output
 IF st_RobotType="ROB1_6620LX_1.90_150" Set SM1_do_Stopped;

 ! aufruf der einzelnen Init Appl / calling the individual Init Appl
 IF n_ApplMax >0 AND n_ApplMax< 31 THEN
   FOR I FROM 1 TO n_ApplMax DO
     IF st_Appl_Info{I,1}="" GOTO END_InitAppl;
     b_ComDummy:=StrToVal(st_Appl_Info{I,1},n_ComDummy);
     %"InitAppl"+NumToStr(n_ComDummy,0)%;
   ENDFOR
 ENDIF
 END_InitAppl:
 ERROR
 !** Error Handler**
 SkipWarn;
 IF ERRNO=ERR_REFUNKPRC TRYNEXT;
ENDPROC !(InitMain)

!*******************************************************************************

PROC JobRequest()
!*************************************************************
!* Befehl Jobanfrage an die SPS / Command Job request to PLC *
!* Trap-Routine                                              *
!*************************************************************
VAR signaldo PLC_JobStarted;
VAR string st_alias2;
CONST string st_C:="PLC_do_Job";
CONST string st_D:="_Started";
!
IF n_JobReqNum>0 THEN
	! Signalnamen erzeugen / signalname to procreate
	IF n_JobReqNum <10 THEN
		st_alias2 :=st_C+"0"+NumToStr(n_JobReqNum,0)+st_D;
	ELSE
		st_alias2 :=st_C+NumToStr(n_JobReqNum,0)+st_D;
	ENDIF
	AliasIO st_alias2, PLC_JobStarted;
	!
  	Set PLC_JobStarted;
ELSE
	! Fehler Jobnum = 0
	ErrWrite \W, "PLC, Trap JobRequest error", "JobNum = 0" ;
ENDIF
n_JobReqNum:=0;
b_JobR_w:=FALSE;
ENDPROC !(JobRequest)

!*******************************************************************************

PROC MoveJ_JobRequest (num Job,  robtarget ToPoint,  speeddata Speed,  zonedata Zone,  PERS tooldata Tool  \PERS wobjdata Wobj)
!*************************************************
!*   Command to call the  job request routine    *
!* synchronous from a joint type motion movement *
!*************************************************
VAR signaldi PLC_JobEnable;
VAR string st_alias;
CONST string st_A:="PLC_di_Job";
CONST string st_B:="_Enable";
! Wert check 1-32
CheckValue Job, 1, 32, 0, "Job Number";
! Signalnamen erzeugen / signalname to procreate
IF Job <10 THEN
	st_alias :=st_A+"0"+NumToStr(Job,0)+st_B;
ELSE
	st_alias :=st_A+NumToStr(Job,0)+st_B;
ENDIF
AliasIO st_alias, PLC_JobEnable;
!
! Programmablaufart pruefen / runmode check
IF (RunMode() = RUN_CONT_CYCLE) AND (PLC_JobEnable=1) AND (Zone <> fine) AND (b_JobR_w = FALSE)THEN
	b_JobR_w:= TRUE;
	n_JobReqNum:=Job;
	! Aufruf von MoveXSync
	MoveJSync ToPoint,Speed,Zone,Tool\WObj?Wobj,"JobRequest";
ELSE
	! Fahre Punkt an
	MoveJ ToPoint,Speed,fine,Tool\WObj?Wobj;

	WHILE PLC_JobEnable=0 DO
      	st_UiHeader:=["Com,Waiting for Job Req ","Com, Warte auf Jobfreigabe ","???"];
    	st_UiHeader_2:=[" from the PLC"," von der SPS","???"];
    	st_UiMsgLine1:=["Waiting for Signal ","Warte auf Signal ","???"];
    	st_UiMsgLine2:=["","","???"];
    	UIMsgBox\Header:=st_UiHeader{n_Sp}+ValToStr(Job)+st_UiHeader_2{n_Sp},st_UiMsgLine1{n_Sp}+st_alias+" = 1"\MsgLine2:=st_UiMsgLine2{n_Sp}
      			\Buttons:=btnNone\Icon:=iconInfo\DIBreak:=PLC_JobEnable;
	ENDWHILE

	! pruefen ob bereits eine Anfrage laeuft
	WaitUntil b_JobR_w = FALSE \PollRate:=0.01;
	!***********************************
	!* Waiting for MoveSync to trigger *
	!***********************************

	n_JobReqNum:=Job;
	JobRequest;
ENDIF
!
BACKWARD
!
MoveJ ToPoint,Speed,fine,Tool\WObj?Wobj;
ERROR
!** Error Handler**
	SkipWarn;
 	IF ERRNO = ERR_TP_DIBREAK TRYNEXT;
ENDPROC !(MoveJ_JobRequest)

!*******************************************************************************

PROC MoveL_JobRequest (num Job,  robtarget ToPoint,  speeddata Speed,  zonedata Zone,  PERS tooldata Tool  \PERS wobjdata Wobj)
!*************************************************
!*   Command to call the  job request routine    *
!* synchronous from a joint type motion movement *
!*************************************************
VAR signaldi PLC_JobEnable;
VAR string st_alias;
CONST string st_A:="PLC_di_Job";
CONST string st_B:="_Enable";
! Wert check 1-32
CheckValue Job, 1, 32, 0, "Job Number";
! Signalnamen erzeugen / signalname to procreate
IF Job <10 THEN
	st_alias :=st_A+"0"+NumToStr(Job,0)+st_B;
ELSE
	st_alias :=st_A+NumToStr(Job,0)+st_B;
ENDIF
AliasIO st_alias, PLC_JobEnable;
!
! Programmablaufart pruefen / runmode check
IF (RunMode() = RUN_CONT_CYCLE) AND (PLC_JobEnable=1) AND (Zone <> fine) AND (b_JobR_w = FALSE)THEN
	b_JobR_w:= TRUE;
	n_JobReqNum:=Job;
	! Aufruf von MoveXSync
	MoveLSync ToPoint,Speed,Zone,Tool\WObj?Wobj,"JobRequest";
ELSE
	! Fahre Punkt an
	MoveL ToPoint,Speed,fine,Tool\WObj?Wobj;

    WHILE PLC_JobEnable=0 DO
      	st_UiHeader:=["Com,Waiting Job Req ","Com, Warte auf Jobfreigabe ","???"];
    	st_UiHeader_2:=[" from the PLC"," von der SPS","???"];
    	st_UiMsgLine1:=["Waiting for Signal ","Warte auf Signal ","???"];
    	st_UiMsgLine2:=["","","???"];
    	UIMsgBox\Header:=st_UiHeader{n_Sp}+ValToStr(Job)+st_UiHeader_2{n_Sp},st_UiMsgLine1{n_Sp}+st_alias+" = 1"\MsgLine2:=st_UiMsgLine2{n_Sp}
      			\Buttons:=btnNone\Icon:=iconInfo\DIBreak:=PLC_JobEnable;
	ENDWHILE

	! pruefen ob bereits eine Anfrage laeuft
	WaitUntil b_JobR_w = FALSE \PollRate:=0.01;
	!***********************************
	!* Waiting for MoveSync to trigger *
	!***********************************

	n_JobReqNum:=Job;
	JobRequest;
ENDIF
!
BACKWARD
!
MoveL ToPoint,Speed,fine,Tool\WObj?Wobj;
ERROR
!** Error Handler**
	SkipWarn;
 	IF ERRNO = ERR_TP_DIBREAK TRYNEXT;
ENDPROC !(MoveL_JobRequest)

!*******************************************************************************

PROC Job_Request (num Job \switch InAdvance )
!*************************************************
!*   Command to call the  job request routine    *
!*          without motion movement              *
!*************************************************
VAR signaldi PLC_JobEnable;
VAR string st_alias;
CONST string st_A:="PLC_di_Job";
CONST string st_B:="_Enable";
VAR errnum err_var;

! Wert check 1-32
CheckValue Job, 1, 32, 0, "Job Number";
! Signalnamen erzeugen / signalname to procreate

IF Job <10 THEN
	st_alias :=st_A+"0"+NumToStr(Job,0)+st_B;
ELSE
	st_alias :=st_A+NumToStr(Job,0)+st_B;
ENDIF

AliasIO st_alias, PLC_JobEnable;

if Present (InAdvance)<>TRUE THEN
    WaitRob\InPos;
    !*****************************
    !* Waiting Robot in position *
    !*****************************
ENDIF

WHILE PLC_JobEnable=0 DO
    st_UiHeader:=["Com,Waiting Job Req ","Com, Warte auf Jobfreigabe ","???"];
    st_UiHeader_2:=[" from the PLC"," von der SPS","???"];
    st_UiMsgLine1:=["Waiting for Signal ","Warte auf Signal ","???"];
    st_UiMsgLine2:=["","","???"];
    UIMsgBox\Header:=st_UiHeader{n_Sp}+ValToStr(Job)+st_UiHeader_2{n_Sp},st_UiMsgLine1{n_Sp}+st_alias+" = 1"\MsgLine2:=st_UiMsgLine2{n_Sp}
    		\Buttons:=btnNone\Icon:=iconInfo\DIBreak:=PLC_JobEnable;
ENDWHILE

n_JobReqNum:=Job;
JobRequest;

BACKWARD

ERROR
!** Error Handler**
	SkipWarn;
 	IF ERRNO = ERR_TP_DIBREAK TRYNEXT;
ENDPROC !(MoveJ_JobRequest)

!*******************************************************************************

PROC Job_Finished (num Job)
!*************************************************
!*   Command to call the  job finished routine   *
!*           without  motion movement            *
!*************************************************

CheckValue Job, 1, 32, 0, "Job Number";

WaitRob\InPos;
!*****************************
!* Waiting Robot in position *
!*****************************

! Ausgang setzen
n_JobFinNum:=Job;
JobFinished;

ENDPROC !(Job_Finished)

!*******************************************************************************

PROC JobFinished()
!***********************************************
!* Job Endemeldung an die SPS 1-32 TrapRoutine *
!*  Job finished communication routine to PLC  *
!***********************************************
VAR signaldo PLC_JobStarted;
VAR signaldo PLC_JobReady;
VAR string st_alias;
VAR string st_alias2;
CONST string st_A:="PLC_do_Job";
CONST string st_B:="_Started";
CONST string st_C:="_Ready";
!
IF n_JobFinNum>0 THEN
	! Signalnamen zusammensetzen
	IF n_JobFinNum <10 THEN
  		st_alias :=st_A+"0"+NumToStr(n_JobFinNum ,0)+st_B;
  		st_alias2 :=st_A+"0"+NumToStr(n_JobFinNum ,0)+st_C;
	ELSE
  		st_alias :=st_A+NumToStr(n_JobFinNum ,0)+st_B;
  		st_alias2 :=st_A+NumToStr(n_JobFinNum ,0)+st_C;
	ENDIF

	! Aliaszuweisen
	AliasIO st_alias, PLC_JobStarted;
	AliasIO st_alias2, PLC_JobReady;

	! Ausgang setzen
	Reset PLC_JobStarted;
	Set PLC_JobReady;
ELSE
  ! Fehler Jobnum = 0
  ErrWrite \W, "PLC, Trap JobFinished error", "JobNum = 0" ;
ENDIF

n_JobFinNum:=0;
b_JobF_w:=FALSE;
ENDPROC !(JobFinished)

!*******************************************************************************

PROC MoveJ_JobFinished (num Job,  robtarget ToPoint,  speeddata Speed,  zonedata Zone,  PERS tooldata Tool  \PERS wobjdata Wobj)
!*************************************************
!*   Command to call the  job finished routine   *
!* synchronous from a joint type motion movement *
!*************************************************
!
CheckValue Job, 1, 32, 0, "Job Number";
!
! Programmablaufart pruefen / runmode check
IF (RunMode() = RUN_CONT_CYCLE) AND (Zone <> fine) AND (b_JobF_w = FALSE)THEN
	b_JobF_w:= TRUE;
	n_JobFinNum:=Job;
	! Aufruf von MoveXSync
	MoveJSync ToPoint,Speed,Zone,Tool\WObj?Wobj,"JobFinished";
ELSE
	! Fahre Punkt an
	MoveJ ToPoint,Speed,fine,Tool\WObj?Wobj;
	! pruefen ob bereits eine Anfrage laeuft
	WaitUntil b_JobF_w = FALSE \PollRate:=0.01;
	! Ausgang setzen
	n_JobFinNum:=Job;
	JobFinished;
ENDIF
!
BACKWARD
!
MoveJ ToPoint,Speed,fine,Tool\WObj?Wobj;
!
ENDPROC !(MoveJ_JobFinished)

!*******************************************************************************

PROC MoveL_JobFinished (num Job, robtarget ToPoint, speeddata Speed, zonedata Zone,  PERS tooldata Tool \PERS wobjdata Wobj)
!**************************************************
!* Command to call the  job finished routine      *
!* synchronous from a Linear type motion movement *
!**************************************************
!
CheckValue Job, 1, 32, 0, "Job Number";
!
! Programmablaufart pruefen / runmode check
IF (RunMode() = RUN_CONT_CYCLE) AND (Zone <> fine) AND (b_JobF_w = FALSE)THEN
	b_JobF_w:= TRUE;
	n_JobFinNum:=Job;
	! Aufruf von MoveXSync
	MoveLSync ToPoint,Speed,Zone,Tool\WObj?Wobj,"JobFinished";
ELSE
	! Fahre Punkt an
	MoveL ToPoint,Speed,fine,Tool\WObj?Wobj;
	! pruefen ob bereits eine Anfrage laeuft
	WaitUntil b_JobF_w = FALSE \PollRate:=0.01;
	! Ausgang setzen
	n_JobFinNum:=Job;
	JobFinished;
ENDIF
!
BACKWARD
!
MoveL ToPoint,Speed,fine,Tool\WObj?Wobj;
!
ENDPROC !(MoveL_JobFinished)

!*******************************************************************************

PROC MoveJ_ProcessComplete (robtarget ToPoint, speeddata Speed, zonedata Zone,  PERS tooldata Tool \PERS wobjdata Wobj)
!*************************************************
!* Command to call the  rocess complete routine  *
!* synchronous from a joint type motion movement *
!*************************************************

! Programmablaufart pruefen / runmode check
IF (RunMode() = RUN_CONT_CYCLE) AND (Zone <> fine) THEN
	MoveJSync ToPoint,Speed,Zone,Tool\WObj?Wobj,"ProcessComplete";
ELSE
	MoveJ ToPoint,Speed,fine,Tool\WObj?Wobj;
    ProcessComplete;
ENDIF

BACKWARD

MoveJ ToPoint,Speed,fine,Tool\WObj?Wobj;

ENDPROC !(MoveJ_ProcessComplete)

!*******************************************************************************

PROC ProcessComplete(\SWITCH  Inpos)
!***************************************************
!*  Process complete communication routine to PLC  *
!***************************************************

IF Present(Inpos) Waittime\InPos,0;

PulseDO\High\PLength:=2.0,PLC_do_Process_Complete;

ENDPROC !(ProcessComplete)

!*******************************************************************************

PROC CollSafetyInit()
!*************************************
!* Intialise Robot collision Control *
!*************************************
  VAR bool b_TimeOut;
  !
  n_CollClZ:=1;
  WaitTime \Inpos, 0.01;
  Reset PLC_do_CollZoneClear;
  Reset PLC_do_CollZoneReq;
  SetGO PLC_go_CollZone, 0;
  ! zum testen mit RobotStudio
  IF NOT RobOS()THEN
    FOR i FROM 1 TO 63 DO
    b_CollZoneOccupied{i}:=FALSE;
  ENDFOR
  RETURN;
  ENDIF ! zum testen mit RobotStudio
  WaitGI PLC_gi_CollZone, 0\MaxTime:=3;
  !********************************************************
  !* Waiting for PLC to set Collision zone number to zero *
  !********************************************************
  !
  WHILE GInput(PLC_gi_CollZone)>0 DO
		st_MsgBoxHeader:=["Com, CollSafetyInit","Com, CollSafetyInit","???"];
		st_MsgBoxLine3:=["Waiting for PLC to send collision zone Nr=0.","Rueckmeldung der Kollisionszone ","???"];
		st_MsgBoxLine4:=["","ist nicht Null","???"];
		st_MsgBoxLine5:=["Check the state at the PLC.","Ueberpruefe den Status an der SPS","???"];
		st_MsgBoxGeraeteName:=["CollSafetyInit","CollSafetyInit","???"];
		n_MsgBoxGeraeteNr:=1;
		st_MsgBoxSignal:="PLC_gi_CollZone";
		st_MsgBoxSignalValue:="0";
		n_MsgBoxApplError:=1;
		n_MsgBoxPLC_Error:=52;
		st_MsgBoxElogLine4:="ComBase/CollSafetyInit";
		MsgBox \diBreakSignal:=SYS_di_ErrReset\ErrorToPLC;
  ENDWHILE
  !
  SetGO PLC_go_CollZone, 63;
  WaitGI PLC_gi_CollZone, 63\MaxTime:=3;
  !******************************************************
  !* Waiting for PLC to set Collision zone number to 63 *
  !******************************************************

  WHILE GInput(PLC_gi_CollZone)<>63 DO
		st_MsgBoxHeader:=["Com, CollSafetyInit","Com, CollSafetyInit","???"];
		st_MsgBoxLine3:=["Waiting for the PLC to send collision zone Nr=63.","Rueckmeldung der Kollisionsschutzzone ","???"];
		st_MsgBoxLine4:=["","ist nicht 63","???"];
		st_MsgBoxLine5:=["Check the state at the PLC.","Ueberpruefe den Status an der SPS","???"];
		st_MsgBoxGeraeteName:=["CollSafetyInit","CollSafetyInit","???"];
		n_MsgBoxGeraeteNr:=1;
		st_MsgBoxSignal:="PLC_gi_CollZone";
		st_MsgBoxSignalValue:="63";
		n_MsgBoxApplError:=2;
		n_MsgBoxPLC_Error:=53;
		st_MsgBoxElogLine4:="ComBase/CollSafetyInit";
		MsgBox \diBreakSignal:=SYS_di_ErrReset\ErrorToPLC;
  ENDWHILE
  !
  Set PLC_do_CollZoneClear;
  !
  WaitDI PLC_di_CollZoneRel,1\MaxTime:=3\TimeFlag:=b_TimeOut;
  !******************************************************
  !* Waiting for Collsion zone release signal from PLC  *
  !******************************************************
  WHILE PLC_di_CollZoneRel=0 DO
		st_MsgBoxHeader:=["Com, CollSafetyInit","Com, CollSafetyInit","???"];
		st_MsgBoxLine3:=["Waiting for Collison Zone release from the PLC.","Kollisionsschutz Strobe","???"];
		st_MsgBoxLine4:=["","ist nicht 1","???"];
		st_MsgBoxLine5:=["Check the state at the PLC.","Ueberpruefe den Status an der SPS","???"];
		st_MsgBoxGeraeteName:=["CollSafetyInit","CollSafetyInit","???"];
		n_MsgBoxGeraeteNr:=1;
		st_MsgBoxSignal:="PLC_di_CollZoneRel";
		st_MsgBoxSignalValue:="1";
		n_MsgBoxApplError:=3;
		n_MsgBoxPLC_Error:=54;
		st_MsgBoxElogLine4:="ComBase/CollSafetyInit";
		MsgBox \diBreakSignal:=SYS_di_ErrReset\ErrorToPLC;
  ENDWHILE
  Reset PLC_do_CollZoneClear;
  !
  SetGO PLC_go_CollZone, 0;
  !
  WaitDI PLC_di_CollZoneRel,0\MaxTime:=3\TimeFlag:=b_TimeOut;
  !***************************************************************
  !* Waiting for Collsion zone release signal from PLC to be off *
  !***************************************************************
  WHILE PLC_di_CollZoneRel=1 DO
		st_MsgBoxHeader:=["Com, CollSafetyInit","Com, CollSafetyInit","???"];
		st_MsgBoxLine3:=["Waiting for collison zone release from PLC to be off.","Kollisionsschutz Strobe","???"];
		st_MsgBoxLine4:=["","ist nicht 0","???"];
		st_MsgBoxLine5:=["Check the state at the PLC.","Ueberpruefe den Status an der SPS","???"];
		st_MsgBoxGeraeteName:=["CollSafetyInit","CollSafetyInit","???"];
		n_MsgBoxGeraeteNr:=1;
		st_MsgBoxSignal:="PLC_di_CollZoneRel";
		st_MsgBoxSignalValue:="0";
		n_MsgBoxApplError:=4;
		n_MsgBoxPLC_Error:=55;
		st_MsgBoxElogLine4:="ComBase/CollSafetyInit";
		MsgBox \diBreakSignal:=SYS_di_ErrReset\ErrorToPLC;
  ENDWHILE
  !
  FOR i FROM 1 TO 63 DO
    b_CollZoneOccupied{i}:=FALSE;
  ENDFOR
  !
  b_CollClearAct:=FALSE;
  !
ERROR
!** Error Handler**
SkipWarn;
IF ERRNO = ERR_WAIT_MAXTIME TRYNEXT;
ENDPROC !(CollSafetyInit)

!*******************************************************************************

PROC CollSafetyRequest(num Coll,String Coll_Descr)
 !*************************************************************
 !* Befehl Anforderung einer Kollisionszone                   *
 !* uebergebene Parameter: num Coll Nummer der Kollisionszone *
 !* Command Collision Zone request Control                    *
 !*************************************************************
 VAR btnres br_UiAnswer;
 VAR bool b_TimeOut;
 VAR errnum errno1;
 VAR Dnum dn_Coll ;

 !Convert Collision zone type num to Dnum
 dn_Coll:=NumToDnum(Coll);

 !ueberpruefung ob schon Angefragt / Check if collision zone already requested

 IF b_CollZoneOccupied{Coll}=TRUE THEN
  	st_MsgBoxHeader:=["Com, CollSafetyRequest Error!","Com, Kollisionsschutzanfrage Fehler!","???"];
	IF OpMode()= OP_MAN_PROG THEN
 		st_UiMsgLine1:=["","","???"];
 		st_UiMsgLine2:=["The ","Fehlerhafte Anfrage fuer ","???"];
		st_UiMsgLine3:=["has already been requested before.","Bereich ist bereits Angefragt! ","???"];
		st_UiMsgLine4:=[" ","ueberpruefe auf eine doppelte Anfrage","???"];
		st_UiMsgLine5:=["Please select 'OK' to continue.","Achtung: Anfragen wird abgebrochen!","???"];

		UIMsgBox\Header:=st_MsgBoxHeader{n_Sp},st_UiMsgLine1{n_Sp}\MsgLine2:=st_UiMsgLine2{n_Sp}+"CollZone= "+NumToStr(Coll,0)
			\MsgLine3:=st_UiMsgLine3{n_Sp}\MsgLine4:=st_UiMsgLine4{n_Sp}\MsgLine5:=st_UiMsgLine5{n_Sp}
			\Buttons:=btnOK\Icon:=iconWarning\Result:=br_UiAnswer;
  	ELSE
     	WHILE b_CollZoneOccupied{Coll}=TRUE DO
     		st_Dummy:=["CollZone= ","CollZone= ","???"];
     		st_Dummy2:=["has been already requested.","bereits angefragt !","???"];
     		st_MsgBoxLine3:=["Incorrect request, only allowed in manual mode.","Fehlerhafte Anfrage kann nur im Handbetrieb und","???"];
			st_MsgBoxLine4:=["Reset the program pointer and","mit neu setzen des Prog.-Zeigers abgebrochen werden.","???"];
			st_MsgBoxLine5:=["check program!","Programmablauf ueberpuefen!!!","???"];
			st_MsgBoxbutton4:=["Ok","Ok","???"];
     		n_MsgBoxApplError:=5;
     		n_MsgBoxPLC_Error:=50;
     		st_MsgBoxElogLine4:="ComBase/CollSafetyRequest";

			MsgBox\diBreakSignal:=SYS_di_ErrReset\Line1:=st_Dummy{n_Sp}+NumToStr(Coll,0)\Line2:=st_Dummy2{n_Sp}\ErrorToPLC;
     	ENDWHILE
   	ENDIF
 ENDIF !b_CollZoneOccupied{Coll}

 !Warten bis vorherige Bearbeitung erledigt\Wait until done prior processing

WaitUntil b_CollClearAct=FALSE\MaxTime:=3\TimeFlag:=b_TimeOut;
!****************************************************
!* Waiting for previous collision clear to complete *
!****************************************************

 WHILE b_CollClearAct=TRUE DO
	st_UiHeader:=["Com, CollZoneClearError","Com, CollZoneClearError","???"];
	st_UiMsgLine2:=["MoveXCollReq: Wait b_CollClearAct=FALSE","MoveXCollReq: Warte auf b_CollClearAct=FALSE","???"];
	st_UiMsgLine3:=["The previous clear function has not been finished yet","Das vorherige Freigeben der Zone ist noch nicht abgeschlossen!","???"];
	UIMsgBox\Header:=st_UiHeader{n_Sp},""\MsgLine2:=st_UiMsgLine2{n_Sp}\MsgLine3:=st_UiMsgLine3{n_Sp}
		\Buttons:=btnNone\Icon:=iconWarning\MaxTime:=1.5\BreakFlag:=errno1;
 ENDWHILE

 CollSafetyComFin;

WHILE  PLC_gi_CollZone<>Coll  OR PLC_di_CollZoneFree<>1 DO
     SetGO PLC_go_CollZone, Coll;

    IF b_ColOption Set PLC_do_CollZoneReq;

     WaitGI PLC_gi_CollZone, Coll\MaxTime:=3;
     !******************************************************
     !*  Waiting for PLC to confirm Collision Zone number  *
     !******************************************************

    !Ensure user string is capped below 41 characters
    IF StrLen(Coll_Descr)>40  Coll_Descr := StrPart(Coll_Descr,1,40);

    IF StrLen(Coll_Descr)>6 THEN
    	st_UiMsgLine4:=["with robots " + Coll_Descr,"mit Robotern" + Coll_Descr,"???"];
    ELSEIF StrLen(Coll_Descr)>2 THEN
    	st_UiMsgLine4:=["with robot " + Coll_Descr,"mit Roboter" + Coll_Descr,"???"];
    ELSE
    	st_UiMsgLine4:=["","","???"];
    ENDIF

     WHILE GInput(PLC_gi_CollZone)<>Coll DO
    	MsgBoxBreak "PLC_gi_CollZone",dn_Coll;

    	st_UiHeader:=["Com, CollSafetyRequest","Com, Kollisionsschutzanfrage","???"];
    	st_UiMsgLine1:=["Waiting for PLC_gi_CollZone = ","Warte auf PLC_gi_CollZone = ","???"];
    	st_UiMsgLine2:=["","","???"];
    	st_UiMsgLine3:=["Waiting for collison zone Nr=","Warte auf angefragte Kollisionszone Nr=","???"];

    	UIMsgBox\Header:=st_UiHeader{n_Sp},st_UiMsgLine1{n_Sp}+NumToStr(Coll,0)\MsgLine2:=st_UiMsgLine2{n_Sp}
    		\MsgLine3:=st_UiMsgLine3{n_Sp}+NumToStr(Coll,0)\MsgLine4:=st_UiMsgLine4{n_Sp}\Buttons:=btnNone\Icon:=iconInfo\diBreak:=VB_di_MsgBoxBrk1\BreakFlag:=errno1;
     ENDWHILE

    Set PLC_do_CollZoneReq;

     WaitDI PLC_di_CollZoneFree,1\MaxTime:=3\TimeFlag:=b_TimeOut;
     !**************************************************
     !* Waiting for Collsion zone Free signal from PLC *
     !**************************************************

     WHILE PLC_di_CollZoneFree=0 DO
    	st_UiHeader:=["Com, CollSafetyRequest","Com, Kollisionsschutzanfrage","???"];
    	st_UiMsgLine1:=["Waiting for collision zone free signal from PLC. PLC_di_CollZoneFree=1","Warte auf  PLC_di_CollZoneFree=1","???"];
    	st_UiMsgLine2:=["","","???"];
    	st_UiMsgLine3:=["The collision zone requested = ","fuer die angefragte Kollisionszone = ","???"];
    	UIMsgBox\Header:=st_UiHeader{n_Sp},MsgLine1:=st_UiMsgLine1{n_Sp}\MsgLine2:=st_UiMsgLine2{n_Sp}\MsgLine3:=st_UiMsgLine3{n_Sp}+NumToStr(Coll,0)
    		\MsgLine4:=st_UiMsgLine4{n_Sp}\Buttons:=btnNone\Icon:=iconInfo\DIBreak:=PLC_di_CollZoneFree\BreakFlag:=errno1;
    ENDWHILE
ENDWHILE

b_CollZoneOccupied{Coll}:=TRUE;

 Reset PLC_do_CollZoneReq;
 SetGO PLC_go_CollZone, 0;

IF b_ColOption <>TRUE THEN
     WaitDI PLC_di_CollZoneFree,0\MaxTime:=3\TimeFlag:=b_TimeOut;
     !************************************************************
     !* Waiting for Collsion zone Free signal from PLC to be off *
     !************************************************************

     WHILE PLC_di_CollZoneFree=1 DO
     	MsgBoxBreak "PLC_di_CollZoneFree",0;

    	st_UiHeader:=["Com, CollSafetyRequest","Com, Kollisionsschutzanfrage","???"];
    	st_UiMsgLine2:=["Waiting for Collision zone free signal to be off. PLC_di_CollZoneFree=0","Warte auf PLC_di_CollZoneFree=0","???"];
    	UIMsgBox\Header:=st_UiHeader{n_Sp},""\MsgLine2:=st_UiMsgLine2{n_Sp}
    		\Buttons:=btnNone\Icon:=iconInfo\diBreak:=VB_di_MsgBoxBrk1\BreakFlag:=errno1;
     ENDWHILE
ENDIF

 ERROR
 !** Error Handler**
 SkipWarn;
 IF ERRNO = ERR_WAIT_MAXTIME TRYNEXT;
 IF ERRNO = ERR_TP_DOBREAK TRYNEXT;
 IF ERRNO = ERR_TP_DIBREAK TRYNEXT;
ENDPROC !(CollSafetyRequest)

!*******************************************************************************

PROC MoveJ_CollReq(  num Coll,  \num Coll_B  \num Coll_C  \num Coll_D  \num Coll_E,  robtarget ToPoint,  speeddata Speed,  zonedata Zone,  PERS tooldata Tool  \PERS wobjdata Wobj\String Coll_Desc\String Coll_Desc_B\String Coll_Desc_C\String Coll_Desc_D\String Coll_Desc_E\switch Conc)
 !***********************************************************************
 !*              Collision zone request with a MoveJ                    *
 !***********************************************************************
 !
 CheckValue Coll, 1, 62, 0, "Coll Number";
 IF Present(Coll_B) CheckValue Coll_B, 1, 62, 0, "Coll Number";
 IF Present(Coll_C) CheckValue Coll_C, 1, 62, 0, "Coll Number";
 IF Present(Coll_D) CheckValue Coll_D, 1, 62, 0, "Coll Number";
 IF Present(Coll_E) CheckValue Coll_E, 1, 62, 0, "Coll Number";

  IF Present (Conc) THEN
    MoveJ\Conc, ToPoint,Speed,Zone,Tool\WObj?Wobj;
 ELSE
    MoveJ ToPoint,Speed,Zone,Tool\WObj?Wobj;
 ENDIF

 IF Present(Coll_Desc) THEN
 	CollSafetyRequest Coll,Coll_Desc;
 ELSE
 	CollSafetyRequest Coll,"";
 ENDIF

 IF Present(Coll_Desc_B) THEN
 	IF Present(Coll_B) CollSafetyRequest Coll_B,Coll_Desc_B;
 ELSE
 	IF Present(Coll_B) CollSafetyRequest Coll_B,"";
 ENDIF

 IF Present(Coll_Desc_C) THEN
 	IF Present(Coll_C) CollSafetyRequest Coll_C,Coll_Desc_C;
 ELSE
 	IF Present(Coll_C) CollSafetyRequest Coll_C,"";
 ENDIF

IF Present(Coll_Desc_D) THEN
 	IF Present(Coll_D) CollSafetyRequest Coll_D,Coll_Desc_D;
ELSE
 	IF Present(Coll_D) CollSafetyRequest Coll_D,"";
ENDIF

IF Present(Coll_Desc_E) THEN
	IF Present(Coll_E) CollSafetyRequest Coll_E,Coll_Desc_E;
ELSE
	IF Present(Coll_E) CollSafetyRequest Coll_E,"";
ENDIF

BACKWARD
 !
 CheckValue Coll, 1, 62, 0, "Coll Number";
 IF Present(Coll_B) CheckValue Coll_B, 1, 62, 0, "Coll Number";
 IF Present(Coll_C) CheckValue Coll_C, 1, 62, 0, "Coll Number";
 IF Present(Coll_D) CheckValue Coll_D, 1, 62, 0, "Coll Number";
 IF Present(Coll_E) CheckValue Coll_E, 1, 62, 0, "Coll Number";
 !
 MoveJ ToPoint,Speed,fine,Tool\WObj?Wobj;
 !
 FOR i FROM 1 TO 5 DO
   n_Coll{i}:=0;
 ENDFOR
 !
 n_CollClZ:=1;
 n_Coll{1}:=Coll;
 !
 IF Present(Coll_B) THEN
   Incr n_CollClZ;
   n_Coll{2}:=Coll_B;
 ENDIF
 !
 IF Present(Coll_C) THEN
   Incr n_CollClZ;
   IF n_Coll{2}=0 THEN
     n_Coll{2}:=Coll_C;
   ELSE
     n_Coll{3}:=Coll_C;
   ENDIF
 ENDIF
 !
 IF Present(Coll_D) THEN
   Incr n_CollClZ;
   IF n_Coll{2}=0 THEN
     n_Coll{2}:=Coll_D;
   ELSE
     IF n_Coll{3}=0 THEN
        n_Coll{3}:=Coll_D;
     ELSE
        n_Coll{4}:=Coll_D;
     ENDIF
   ENDIF
 ENDIF
 !
 IF Present(Coll_E) THEN
   Incr n_CollClZ;
   IF n_Coll{2}=0 THEN
     n_Coll{2}:=Coll_E;
   ELSE
     IF n_Coll{3}=0 THEN
       n_Coll{3}:=Coll_E;
     ELSE
       IF n_Coll{4}=0 THEN
         n_Coll{4}:=Coll_E;
       ELSE
         n_Coll{5}:=Coll_E;
       ENDIF
     ENDIF
   ENDIF
 ENDIF
 !
 CollSafetyClear;
 !
ENDPROC !(MoveJ_CollReq)

!*******************************************************************************

PROC MoveL_CollReq(  num Coll,  \num Coll_B  \num Coll_C  \num Coll_D  \num Coll_E,  robtarget ToPoint,  speeddata Speed,  zonedata Zone,  PERS tooldata Tool  \PERS wobjdata Wobj\String Coll_Desc\String Coll_Desc_B\String Coll_Desc_C\String Coll_Desc_D\String Coll_Desc_E\switch Conc)
 !*********************************************************
 !*                  Befehl MoveL_CollClr                 *
 !*  Command MoveL with Triggering of CollSafety Request  *
 !*********************************************************
 CheckValue Coll, 1, 62, 0, "Coll Number";
 IF Present(Coll_B) CheckValue Coll_B, 1, 62, 0, "Coll Number";
 IF Present(Coll_C) CheckValue Coll_C, 1, 62, 0, "Coll Number";
 IF Present(Coll_D) CheckValue Coll_D, 1, 62, 0, "Coll Number";
 IF Present(Coll_E) CheckValue Coll_E, 1, 62, 0, "Coll Number";

 IF Present (Conc) THEN
    MoveL\Conc, ToPoint,Speed,Zone,Tool\WObj?Wobj;
 ELSE
    MoveL ToPoint,Speed,Zone,Tool\WObj?Wobj;
 ENDIF

 IF Present(Coll_Desc) THEN
 	CollSafetyRequest Coll,Coll_Desc;
 ELSE
 	CollSafetyRequest Coll,"";
 ENDIF

 IF Present(Coll_Desc_B) THEN
 	IF Present(Coll_B) CollSafetyRequest Coll_B,Coll_Desc_B;
 ELSE
 	IF Present(Coll_B) CollSafetyRequest Coll_B,"";
 ENDIF

 IF Present(Coll_Desc_C) THEN
 	IF Present(Coll_C) CollSafetyRequest Coll_C,Coll_Desc_C;
 ELSE
 	IF Present(Coll_C) CollSafetyRequest Coll_C,"";
 ENDIF

IF Present(Coll_Desc_D) THEN
 	IF Present(Coll_D) CollSafetyRequest Coll_D,Coll_Desc_D;
ELSE
 	IF Present(Coll_D) CollSafetyRequest Coll_D,"";
ENDIF

IF Present(Coll_Desc_E) THEN
	IF Present(Coll_E) CollSafetyRequest Coll_E,Coll_Desc_E;
ELSE
	IF Present(Coll_E) CollSafetyRequest Coll_E,"";
ENDIF

 BACKWARD
 !
 CheckValue Coll, 1, 62, 0, "Coll Number";
 IF Present(Coll_B) CheckValue Coll_B, 1, 62, 0, "Coll Number";
 IF Present(Coll_C) CheckValue Coll_C, 1, 62, 0, "Coll Number";
 IF Present(Coll_D) CheckValue Coll_D, 1, 62, 0, "Coll Number";
 IF Present(Coll_E) CheckValue Coll_E, 1, 62, 0, "Coll Number";
 !
 MoveL ToPoint,Speed,fine,Tool\WObj?Wobj;
 !
 FOR i FROM 1 TO 5 DO
   n_Coll{i}:=0;
 ENDFOR
 !
 n_CollClZ:=1;
 n_Coll{1}:=Coll;
 !
 IF Present(Coll_B) THEN
   Incr n_CollClZ;
   n_Coll{2}:=Coll_B;
 ENDIF
 !
 IF Present(Coll_C) THEN
   Incr n_CollClZ;
   IF n_Coll{2}=0 THEN
     n_Coll{2}:=Coll_C;
   ELSE
     n_Coll{3}:=Coll_C;
   ENDIF
 ENDIF
 !
 IF Present(Coll_D) THEN
   Incr n_CollClZ;
   IF n_Coll{2}=0 THEN
     n_Coll{2}:=Coll_D;
   ELSE
     IF n_Coll{3}=0 THEN
       n_Coll{3}:=Coll_D;
     ELSE
       n_Coll{4}:=Coll_D;
     ENDIF
   ENDIF
 ENDIF
 !
 IF Present(Coll_E) THEN
   Incr n_CollClZ;
   IF n_Coll{2}=0 THEN
     n_Coll{2}:=Coll_E;
   ELSE
     IF n_Coll{3}=0 THEN
       n_Coll{3}:=Coll_E;
     ELSE
       IF n_Coll{4}=0 THEN
         n_Coll{4}:=Coll_E;
       ELSE
         n_Coll{5}:=Coll_E;
       ENDIF
     ENDIF
   ENDIF
 ENDIF
 !
 CollSafetyClear;
 !
ENDPROC !(MoveL_CollReq)

!*******************************************************************************

PROC Coll_Request(  num Coll,  \num Coll_B  \num Coll_C  \num Coll_D  \num Coll_E,String Coll_Desc\String Coll_Desc_B\String Coll_Desc_C\String Coll_Desc_D\String Coll_Desc_E)
 !***********************************************************************
 !*          Collision zone request without motion points               *
 !***********************************************************************

 CheckValue Coll, 1, 62, 0, "Coll Number";
 IF Present(Coll_B) CheckValue Coll_B, 1, 62, 0, "Coll Number";
 IF Present(Coll_C) CheckValue Coll_C, 1, 62, 0, "Coll Number";
 IF Present(Coll_D) CheckValue Coll_D, 1, 62, 0, "Coll Number";
 IF Present(Coll_E) CheckValue Coll_E, 1, 62, 0, "Coll Number";

 IF Present(Coll_Desc) THEN
 	CollSafetyRequest Coll,Coll_Desc;
 ELSE
 	CollSafetyRequest Coll,"";
 ENDIF

 IF Present(Coll_Desc_B) THEN
 	IF Present(Coll_B) CollSafetyRequest Coll_B,Coll_Desc_B;
 ELSE
 	IF Present(Coll_B) CollSafetyRequest Coll_B,"";
 ENDIF

 IF Present(Coll_Desc_C) THEN
 	IF Present(Coll_C) CollSafetyRequest Coll_C,Coll_Desc_C;
 ELSE
 	IF Present(Coll_C) CollSafetyRequest Coll_C,"";
 ENDIF

IF Present(Coll_Desc_D) THEN
 	IF Present(Coll_D) CollSafetyRequest Coll_D,Coll_Desc_D;
ELSE
 	IF Present(Coll_D) CollSafetyRequest Coll_D,"";
ENDIF

IF Present(Coll_Desc_E) THEN
	IF Present(Coll_E) CollSafetyRequest Coll_E,Coll_Desc_E;
ELSE
	IF Present(Coll_E) CollSafetyRequest Coll_E,"";
ENDIF

BACKWARD

 CheckValue Coll, 1, 62, 0, "Coll Number";
 IF Present(Coll_B) CheckValue Coll_B, 1, 62, 0, "Coll Number";
 IF Present(Coll_C) CheckValue Coll_C, 1, 62, 0, "Coll Number";
 IF Present(Coll_D) CheckValue Coll_D, 1, 62, 0, "Coll Number";
 IF Present(Coll_E) CheckValue Coll_E, 1, 62, 0, "Coll Number";

  FOR i FROM 1 TO 5 DO
   n_Coll{i}:=0;
 ENDFOR

 n_CollClZ:=1;
 n_Coll{1}:=Coll;

 IF Present(Coll_B) THEN
   Incr n_CollClZ;
   n_Coll{2}:=Coll_B;
 ENDIF

 IF Present(Coll_C) THEN
   Incr n_CollClZ;
   IF n_Coll{2}=0 THEN
     n_Coll{2}:=Coll_C;
   ELSE
     n_Coll{3}:=Coll_C;
   ENDIF
 ENDIF

 IF Present(Coll_D) THEN
   Incr n_CollClZ;
   IF n_Coll{2}=0 THEN
     n_Coll{2}:=Coll_D;
   ELSE
     IF n_Coll{3}=0 THEN
        n_Coll{3}:=Coll_D;
     ELSE
        n_Coll{4}:=Coll_D;
     ENDIF
   ENDIF
 ENDIF

 IF Present(Coll_E) THEN
   Incr n_CollClZ;
   IF n_Coll{2}=0 THEN
     n_Coll{2}:=Coll_E;
   ELSE
     IF n_Coll{3}=0 THEN
       n_Coll{3}:=Coll_E;
     ELSE
       IF n_Coll{4}=0 THEN
         n_Coll{4}:=Coll_E;
       ELSE
         n_Coll{5}:=Coll_E;
       ENDIF
     ENDIF
   ENDIF
 ENDIF

 CollSafetyClear;

ENDPROC !(Coll_Request)

!*******************************************************************************

PROC CollSafetyComFin()
 !*************************************************************
 !*  Prozedur Kollisions Kommunikation mit SPS abgearbeitet   *
 !*            uebergebene Parameter: keine                   *
 !*            Collision Zone Control Complete                *
 !*************************************************************
 VAR bool b_TimeOut;
 VAR errnum errno1;

 !Request beendet\Request completed
 WaitDO PLC_do_CollZoneReq,0\MaxTime:=3\TimeFlag:=b_TimeOut;
 !*************************************************************
 !* Waiting for Collsion zone Requset output to PLC to be off *
 !*************************************************************

 WHILE DOutput(PLC_do_CollZoneReq)=1 DO
 	MsgBoxBreak "PLC_do_CollZoneReq",0;

	st_UiHeader:=["Com, CollSafetyComFin","Com, CollSafetyComFin","???"];
	st_UiMsgLine2:=["Waiting for Collision Zone Request output to be off. PLC_do_CollZoneReq=0","Warte auf PLC_do_CollZoneReq=0","???"];
	UIMsgBox\Header:=st_UiHeader{n_Sp},""\MsgLine2:=st_UiMsgLine2{n_Sp}
		\Buttons:=btnNone\Icon:=iconInfo\DIBreak:=VB_di_MsgBoxBrk1\BreakFlag:=errno1;
 ENDWHILE

 WaitDI PLC_di_CollZoneFree,0\MaxTime:=3\TimeFlag:=b_TimeOut;
 !************************************************************
 !* Waiting for Collsion zone Free signal from PLC to be off *
 !************************************************************

 WHILE PLC_di_CollZoneFree=1 DO
 	MsgBoxBreak "PLC_di_CollZoneFree",0;

	st_UiHeader:=["Com, CollSafetyComFin","Com, CollSafetyComFin","???"];
	st_UiMsgLine2:=["Waiting for collision zone free from PLC to be off. PLC_di_CollZoneFree=0","Warte auf PLC_di_CollZoneFree=0","???"];
	UIMsgBox\Header:=st_UiHeader{n_Sp}, ""\MsgLine2:=st_UiMsgLine2{n_Sp}\Buttons:=btnNone\Icon:=iconInfo\DIBreak:=VB_di_MsgBoxBrk1\BreakFlag:=errno1;
 ENDWHILE

 !Clear beendet / Clear finished
 WaitDO PLC_do_CollZoneClear,0\MaxTime:=3\TimeFlag:=b_TimeOut;
 !*************************************************************
 !* Waiting for Collsion zone Clear signal from PLC to be off *
 !*************************************************************

 WHILE DOutput(PLC_do_CollZoneClear)=1 DO
 	MsgBoxBreak "PLC_do_CollZoneClear",0;

	st_UiHeader:=["Com, CollSafetyComFin","Com, CollSafetyComFin","???"];
	st_UiMsgLine2:=["Waiting for collision zone clear from PLC to be off. PLC_do_CollZoneClear=0","Warte auf PLC_do_CollZoneClear=0","???"];
	UIMsgBox\Header:=st_UiHeader{n_Sp},""\MsgLine2:=st_UiMsgLine2{n_Sp}
		\Buttons:=btnNone\Icon:=iconInfo\MaxTime:=1\DIBreak:=VB_di_MsgBoxBrk1\BreakFlag:=errno1;
 ENDWHILE

 WaitDI PLC_di_CollZoneRel,0\MaxTime:=3\TimeFlag:=b_TimeOut;
 !***************************************************************
 !* Waiting for Collsion zone Release signal from PLC to be off *
 !***************************************************************

 WHILE PLC_di_CollZoneRel=1 DO
 	MsgBoxBreak "PLC_di_CollZoneRel",0;

	st_UiHeader:=["Com, CollSafetyComFin","Com, CollSafetyComFin","???"];
	st_UiMsgLine2:=["Waiting for collision zone release from PLC to be off. PLC_di_CollZoneRel=0","Warte auf PLC_di_CollZoneRel=0","???"];
	UIMsgBox\Header:=st_UiHeader{n_Sp},""\MsgLine2:=st_UiMsgLine2{n_Sp}
		\Buttons:=btnNone\Icon:=iconInfo\MaxTime:=1\DIBreak:=VB_di_MsgBoxBrk1\BreakFlag:=errno1;
 ENDWHILE

 WaitGI PLC_gi_CollZone, 0\MaxTime:=3;
 !********************************************************
 !* Waiting for PLC to set Collision zone number to zero *
 !********************************************************

 WHILE GInput(PLC_gi_CollZone)>0 DO
 	MsgBoxBreak "PLC_gi_CollZone",0;

	st_UiHeader:=["Com, CollSafetyComFin","Com, CollSafetyComFin","???"];
	st_UiMsgLine2:=["Waiting for PLC to send collision zone zero. PLC_gi_CollZone=0","Warte auf PLC_gi_CollZone=0","???"];
	UIMsgBox\Header:=st_UiHeader{n_Sp},""\MsgLine2:=st_UiMsgLine2{n_Sp}\Buttons:=btnNone\Icon:=iconInfo\diBreak:=VB_di_MsgBoxBrk1\BreakFlag:=errno1;
 ENDWHILE
 !
 ERROR
 !** Error Handler**
 SkipWarn;
 IF ERRNO = ERR_WAIT_MAXTIME TRYNEXT;
 IF ERRNO = ERR_TP_DIBREAK TRYNEXT;

ENDPROC !(CollSafetyComFin)

!*******************************************************************************

PROC CollClearAll()
  !****************************************
  !* Init Zonen / Init zone               *
  !* alle Zonen loeschen / clear all zone *
  !****************************************
  WaitRob \InPos;
  CollSafetyInit;
ENDPROC !(CollClearAll)

!*******************************************************************************

PROC CollSafetyClear()
 !*************************************************************
 !*          Prozedur Freigabe einer Kollisionszone           *
 !*            uebergebene Parameter: keine                   *
 !*            Collision Zone Control Clear                   *
 !*************************************************************
 VAR bool b_TimeOut;
 VAR errnum errno1;

CollSafetyComFin;

 FOR i FROM 1 TO n_CollClZ DO
    !Kein abloeschen wenn nicht angefordert

    WaitDI PLC_di_CollZoneRel,0\MaxTime:=3\TimeFlag:=b_TimeOut;
    !***************************************************************
    !* Waiting for Collsion zone release signal from PLC to be off *
    !***************************************************************

    WHILE PLC_di_CollZoneRel=1 DO
    	st_UiHeader:=["Com, CollSafetyClear","Com, CollSafetyClear","???"];
    	st_UiMsgLine2:=["Waiting for collision zone release from PLC to be off. PLC_di_CollZoneRel = 0","Warte auf PLC_di_CollZoneRel = 0","???"];
    	UIMsgBox\Header:=st_UiHeader{n_Sp},""\MsgLine2:=st_UiMsgLine2{n_Sp}\Buttons:=btnNone\Icon:=iconInfo\MaxTime:=1\BreakFlag:=errno1;
    ENDWHILE

    IF b_CollZoneOccupied{n_Coll{i}}=TRUE THEN
        WHILE PLC_gi_CollZone<> n_Coll{i} OR PLC_di_CollZoneRel<>1 DO

            SetGO PLC_go_CollZone, n_Coll{i};

            IF b_ColOption Set PLC_do_CollZoneClear;

            WaitGI PLC_gi_CollZone, n_Coll{i}\MaxTime:=3;
            !******************************************************
            !*  Waiting for PLC to confirm Collision Zone number  *
            !******************************************************

            WHILE GInput(PLC_gi_CollZone)<>n_Coll{i} DO
                st_UiHeader:=["Com, CollSafetyClear","Com, CollSafetyClear","???"];
                st_UiMsgLine2:=["Waiting for PLC to echo back collision zone number. PLC_gi_CollZone = ","Warte auf PLC_gi_CollZone = ","???"];
                UIMsgBox\Header:=st_UiHeader{n_Sp},""\MsgLine2:=st_UiMsgLine2{n_Sp}+NumToStr(n_Coll{i},0)\Buttons:=btnNone\Icon:=iconInfo\MaxTime:=1\BreakFlag:=errno1;
            ENDWHILE

            Set PLC_do_CollZoneClear;

            WaitDI PLC_di_CollZoneRel,1\MaxTime:=3\TimeFlag:=b_TimeOut;
            !******************************************************
            !* Waiting for Collsion zone release signal from PLC  *
            !******************************************************

            WHILE PLC_di_CollZoneRel=0 DO
                st_UiHeader:=["Com, CollSafetyClear","Com, CollSafetyClear","???"];
                st_UiMsgLine2:=["Waiting for collison zone release from PLC. PLC_di_CollZoneRel = 1","Warte auf PLC_di_CollZoneRel = 1","???"];
                UIMsgBox\Header:=st_UiHeader{n_Sp},""\MsgLine2:=st_UiMsgLine2{n_Sp}\Buttons:=btnNone\Icon:=iconInfo\MaxTime:=1\BreakFlag:=errno1;
            ENDWHILE
        ENDWHILE

        b_CollZoneOccupied{n_Coll{i}}:=FALSE;

    ENDIF

    Reset PLC_do_CollZoneClear;
    SetGO PLC_go_CollZone, 0;

    IF b_ColOption <>TRUE THEN
         WaitDI PLC_di_CollZoneRel,0\MaxTime:=3\TimeFlag:=b_TimeOut;
         !***************************************************************
         !* Waiting for Collsion zone release signal from PLC to be off *
         !***************************************************************

         WHILE PLC_di_CollZoneRel=1 DO
        	st_UiHeader:=["Com, CollSafetyClear","Com, CollSafetyClear","???"];
        	st_UiMsgLine2:=["Waiting for collision zone release from PLC to be off. PLC_di_CollZoneRel = 0","Warte auf PLC_di_CollZoneRel = 0","???"];
        	UIMsgBox\Header:=st_UiHeader{n_Sp},""\MsgLine2:=st_UiMsgLine2{n_Sp}\Buttons:=btnNone\Icon:=iconInfo\MaxTime:=1\BreakFlag:=errno1;
         ENDWHILE
    ENDIF
 ENDFOR

 b_CollClearAct:=FALSE;
 ERROR
 !** Error Handler**
 SkipWarn;
 IF ERRNO = ERR_WAIT_MAXTIME TRYNEXT;
ENDPROC !(CollSafetyClear)
!*******************************************************************************

PROC Coll_Clear(num Coll  \num Coll_B  \num Coll_C  \num Coll_D  \num Coll_E)
 !***************************
 !*    Befehl MoveJ_CollClr *
 !*   without motion points *
 !***************************

 VAR btnres br_UiAnswer;
 VAR bool b_TimeOut;
 VAR errnum errno1;

 CheckValue Coll, 1, 62, 0, "Coll Number";
 IF Present(Coll_B) CheckValue Coll_B, 1, 62, 0, "Coll Number";
 IF Present(Coll_C) CheckValue Coll_C, 1, 62, 0, "Coll Number";
 IF Present(Coll_D) CheckValue Coll_D, 1, 62, 0, "Coll Number";
 IF Present(Coll_E) CheckValue Coll_E, 1, 62, 0, "Coll Number";

 !Warten bis vorherige Bearbeitung erledigt

 WaitUntil b_CollClearAct=FALSE\MaxTime:=3\TimeFlag:=b_TimeOut;
 !*************************************************************
 !*   Waiting for acknowledge that the Collsion was released  *
 !*************************************************************

 IF b_CollClearAct=TRUE THEN
   IF OpMode()= OP_MAN_PROG THEN
     st_UiHeader:=["Com, CollZoneClearError","Com, CollZoneClearError","???"];
     st_UiMsgLine1:=["Warning","Achtung","???"];
     st_UiMsgLine2:=["","","???"];
     st_UiMsgLine3:=["The clear collision zone routine was interrupted!","Die Funktion loesche Kollisionsschutz wurde abgebrochen","???"];
     st_UiMsgLine4:=["Please confirm in Manual Mode! ","Betaetigen in Handbetrieb","???"];
	UIMsgBox\Header:=st_UiHeader{n_Sp},st_UiMsgLine1{n_Sp}\MsgLine2:=st_UiMsgLine2{n_Sp}
  		\MsgLine3:=st_UiMsgLine3{n_Sp}\MsgLine4:=st_UiMsgLine4{n_Sp}
	 	\Buttons:=btnOK\Icon:=iconError;
     b_CollClearAct:=FALSE;
     TPErase;
     TPShow TP_LATEST;
   ELSE
     WHILE b_CollClearAct=TRUE DO
		st_UiHeader:=["Com, CollZoneClearError","Com, CollZoneClearError","???"];
		st_UiMsgLine2:=["Coll_Clear: Wait b_CollClearAct=FALSE","Coll_Clear: Warte auf b_CollClearAct=FALSE","???"];
		st_UiMsgLine3:=["The clear function has not been finished yet","Das Freigeben der Zone ist noch nicht abgeschlossen!","???"];
		UIMsgBox\Header:=st_UiHeader{n_Sp},""\MsgLine2:=st_UiMsgLine2{n_Sp}\MsgLine3:=st_UiMsgLine3{n_Sp}
			\Buttons:=btnNone\Icon:=iconWarning\MaxTime:=1\BreakFlag:=errno1;
     ENDWHILE
   ENDIF
 ENDIF

 !In bearbeitung
 b_CollClearAct:=TRUE;

 !Init Zonen / Init zone
 FOR i FROM 1 TO 5 DO
   n_Coll{i}:=0;
 ENDFOR

 !Einlesen der Zonen / Reading the Zone
 n_CollClZ:=1;
 n_Coll{1}:=Coll;

IF Present(Coll_B) THEN
    Incr n_CollClZ;
    n_Coll{2}:=Coll_B;
ENDIF

IF Present(Coll_C) THEN
    Incr n_CollClZ;
    IF n_Coll{2}=0 THEN
        n_Coll{2}:=Coll_C;
    ELSE
        n_Coll{3}:=Coll_C;
    ENDIF
ENDIF

IF Present(Coll_D) THEN
    Incr n_CollClZ;
    IF n_Coll{2}=0 THEN
        n_Coll{2}:=Coll_D;
    ELSE
        IF n_Coll{3}=0 THEN
            n_Coll{3}:=Coll_D;
        ELSE
            n_Coll{4}:=Coll_D;
        ENDIF
    ENDIF
ENDIF

IF Present(Coll_E) THEN
    Incr n_CollClZ;
    IF n_Coll{2}=0 THEN
        n_Coll{2}:=Coll_E;
    ELSE
        IF n_Coll{3}=0 THEN
            n_Coll{3}:=Coll_E;
        ELSE
            IF n_Coll{4}=0 THEN
                n_Coll{4}:=Coll_E;
            ELSE
                n_Coll{5}:=Coll_E;
            ENDIF
        ENDIF
    ENDIF
ENDIF

 !Wenn nicht besetzt / When not occupied
 FOR i FROM 1 TO n_CollClZ DO
   IF OpMode()= OP_AUTO THEN
     WHILE b_CollZoneOccupied{n_Coll{i}}=FALSE DO
		st_MsgBoxHeader:=["Com, MoveLCollClr","Com, Kollisionsschutzfreigabe","Com,???"];
		st_Dummy:=["CollZone= "+NumToStr(n_Coll{i},0),"CollZone= "+NumToStr(n_Coll{i},0),"???"];
		st_Dummy2:=["is not already requested!","war nicht angefragt!","???"];
		st_MsgBoxbutton4:=["Ok","Ok","???"];
		st_MsgBoxbutton5:=["","","???"];
		n_MsgBoxApplError:=0;
		n_MsgBoxPLC_Error:=51;
		st_MsgBoxElogLine4:="ComBase/MoveLCollClr";
		MsgBox\diBreakSignal:=SYS_di_ErrReset\Line1:=st_Dummy{n_Sp}\Line2:=st_Dummy2{n_Sp}\ErrorToPLC;
     ENDWHILE
   ELSE
     IF b_CollZoneOccupied{n_Coll{i}}=FALSE THEN
       st_UiHeader:=["Com, MoveLCollClr","Com, Kollisionsschutzfreigabe","???"];
		st_UiMsgLine1:=["Clear Error","Freigabefehler!","???"];
		st_UiMsgLine2:=["is not already requested!","Bereich war nicht angefragt!","???"];
		st_UiMsgLine3:=["Please check the collisions zones already","ueberpruefe den Status der Kollisionszone","???"];
		st_UiMsgLine4:=["requested and confirm their status. ","Bestaetige den Zustand !","???"];
		UIMsgBox\Header:=st_UiHeader{n_Sp},st_UiMsgLine1{n_Sp}\MsgLine2:=st_UiMsgLine2{n_Sp}
  		\MsgLine3:=st_UiMsgLine3{n_Sp}\MsgLine4:=st_UiMsgLine4{n_Sp}
	 	\Buttons:=btnOK\Icon:=iconWarning;
     ENDIF
   ENDIF
 ENDFOR

WaitRob\InPos;
!*****************************
!* Waiting Robot in position *
!*****************************

CollSafetyClear;

BACKWARD

 CheckValue Coll, 1, 62, 0, "Coll Number";
 IF Present(Coll_B) CheckValue Coll_B, 1, 62, 0, "Coll Number";
 IF Present(Coll_C) CheckValue Coll_C, 1, 62, 0, "Coll Number";
 IF Present(Coll_D) CheckValue Coll_D, 1, 62, 0, "Coll Number";
 IF Present(Coll_E) CheckValue Coll_E, 1, 62, 0, "Coll Number";

 CollSafetyRequest Coll,"";
 IF Present(Coll_B) CollSafetyRequest Coll_B,"";
 IF Present(Coll_C) CollSafetyRequest Coll_C,"";
 IF Present(Coll_D) CollSafetyRequest Coll_D,"";
 IF Present(Coll_E) CollSafetyRequest Coll_E,"";

 ERROR
 !** Error Handler**
 SkipWarn;
 IF ERRNO = ERR_WAIT_MAXTIME TRYNEXT;
ENDPROC !(Coll_Clear)

!*******************************************************************************

PROC MoveJ_CollClr(  num Coll  \num Coll_B  \num Coll_C  \num Coll_D  \num Coll_E,  robtarget ToPoint,  speeddata Speed,  zonedata Zone,  PERS tooldata Tool  \PERS wobjdata Wobj)
 !*********************************************************
 !*                  Befehl MoveJ_CollClr                 *
 !*   Command MoveJ with Triggering of CollSafety Clear   *
 !*********************************************************
 VAR btnres br_UiAnswer;
 VAR bool b_TimeOut;
 VAR errnum errno1;
 !
 CheckValue Coll, 1, 62, 0, "Coll Number";
 IF Present(Coll_B) CheckValue Coll_B, 1, 62, 0, "Coll Number";
 IF Present(Coll_C) CheckValue Coll_C, 1, 62, 0, "Coll Number";
 IF Present(Coll_D) CheckValue Coll_D, 1, 62, 0, "Coll Number";
 IF Present(Coll_E) CheckValue Coll_E, 1, 62, 0, "Coll Number";
 !
 !Warten bis vorherige Bearbeitung erledigt
 !
 WaitUntil b_CollClearAct=FALSE\MaxTime:=3\TimeFlag:=b_TimeOut;
 !*************************************************************
 !*   Waiting for acknowledge that the Collsion was released  *
 !*************************************************************
 IF b_CollClearAct=TRUE THEN
   IF OpMode()= OP_MAN_PROG THEN
     st_UiHeader:=["Com, CollZoneClearError","Com, CollZoneClearError","???"];
     st_UiMsgLine1:=["Warning","Achtung","???"];
     st_UiMsgLine2:=["","","???"];
     st_UiMsgLine3:=["The clear collision zone routine was interrupted!","Die Funktion loesche Kollisionsschutz wurde abgebrochen","???"];
     st_UiMsgLine4:=["Please confirm in Manual Mode! ","Betaetigen in Handbetrieb","???"];
	UIMsgBox\Header:=st_UiHeader{n_Sp},st_UiMsgLine1{n_Sp}\MsgLine2:=st_UiMsgLine2{n_Sp}
  		\MsgLine3:=st_UiMsgLine3{n_Sp}\MsgLine4:=st_UiMsgLine4{n_Sp}
	 	\Buttons:=btnOK\Icon:=iconError;
     b_CollClearAct:=FALSE;
     TPErase;
     TPShow TP_LATEST;
   ELSE
     WHILE b_CollClearAct=TRUE DO
		st_UiHeader:=["Com, CollZoneClearError","Com, CollZoneClearError","???"];
		st_UiMsgLine2:=["MoveJCollClr: Wait b_CollClearAct=FALSE","MoveJCollClr: Warte auf b_CollClearAct=FALSE","???"];
		st_UiMsgLine3:=["The clear function has not been finished yet","Das Freigeben der Zone ist noch nicht abgeschlossen!","???"];
		UIMsgBox\Header:=st_UiHeader{n_Sp},""\MsgLine2:=st_UiMsgLine2{n_Sp}\MsgLine3:=st_UiMsgLine3{n_Sp}
			\Buttons:=btnNone\Icon:=iconWarning\MaxTime:=1\BreakFlag:=errno1;
     ENDWHILE
   ENDIF
 ENDIF
 !
 !In bearbeitung
 b_CollClearAct:=TRUE;
 !
 !Init Zonen / Init zone
 !
 FOR i FROM 1 TO 5 DO
   n_Coll{i}:=0;
 ENDFOR
 !
 !Einlesen der Zonen / Reading the Zone
 !
 n_CollClZ:=1;
 n_Coll{1}:=Coll;
 !
 IF Present(Coll_B) THEN
   Incr n_CollClZ;
   n_Coll{2}:=Coll_B;
 ENDIF
 !
 IF Present(Coll_C) THEN
   Incr n_CollClZ;
   IF n_Coll{2}=0 THEN
     n_Coll{2}:=Coll_C;
   ELSE
     n_Coll{3}:=Coll_C;
   ENDIF
 ENDIF
 !
 IF Present(Coll_D) THEN
   Incr n_CollClZ;
   IF n_Coll{2}=0 THEN
     n_Coll{2}:=Coll_D;
   ELSE
     IF n_Coll{3}=0 THEN
       n_Coll{3}:=Coll_D;
     ELSE
       n_Coll{4}:=Coll_D;
     ENDIF
   ENDIF
 ENDIF
 !
 IF Present(Coll_E) THEN
   Incr n_CollClZ;
   IF n_Coll{2}=0 THEN
     n_Coll{2}:=Coll_E;
   ELSE
     IF n_Coll{3}=0 THEN
       n_Coll{3}:=Coll_E;
     ELSE
       IF n_Coll{4}=0 THEN
         n_Coll{4}:=Coll_E;
       ELSE
         n_Coll{5}:=Coll_E;
       ENDIF
     ENDIF
   ENDIF
 ENDIF
 !
 !Wenn nicht besetzt / When not occupied
 !
 FOR i FROM 1 TO n_CollClZ DO
   IF OpMode()= OP_AUTO THEN
     WHILE b_CollZoneOccupied{n_Coll{i}}=FALSE DO
		st_MsgBoxHeader:=["Com, MoveLCollClr","Com, Kollisionsschutzfreigabe","Com,???"];
		st_Dummy:=["CollZone= "+NumToStr(n_Coll{i},0),"CollZone= "+NumToStr(n_Coll{i},0),"???"];
		st_Dummy2:=["is not already requested!","war nicht angefragt!","???"];
		st_MsgBoxbutton4:=["Ok","Ok","???"];
		st_MsgBoxbutton5:=["","","???"];
		n_MsgBoxApplError:=0;
		n_MsgBoxPLC_Error:=51;
		st_MsgBoxElogLine4:="ComBase/MoveLCollClr";
		MsgBox\diBreakSignal:=SYS_di_ErrReset\Line1:=st_Dummy{n_Sp}\Line2:=st_Dummy2{n_Sp}\ErrorToPLC;
     ENDWHILE
   ELSE
     IF b_CollZoneOccupied{n_Coll{i}}=FALSE THEN
       st_UiHeader:=["Com, MoveLCollClr","Com, Kollisionsschutzfreigabe","???"];
		st_UiMsgLine1:=["Clear Error","Freigabefehler!","???"];
		st_UiMsgLine2:=["is not already requested!","Bereich war nicht angefragt!","???"];
		st_UiMsgLine3:=["Please check the collisions zones already","ueberpruefe den Status der Kollisionszone","???"];
		st_UiMsgLine4:=["requested and confirm their status. ","Bestaetige den Zustand !","???"];
		UIMsgBox\Header:=st_UiHeader{n_Sp},st_UiMsgLine1{n_Sp}\MsgLine2:=st_UiMsgLine2{n_Sp}
  		\MsgLine3:=st_UiMsgLine3{n_Sp}\MsgLine4:=st_UiMsgLine4{n_Sp}
	 	\Buttons:=btnOK\Icon:=iconWarning;
     ENDIF
   ENDIF
 ENDFOR

 IF RunMode() = RUN_CONT_CYCLE THEN
   MoveJSync ToPoint,Speed, Zone,Tool\WObj?Wobj, "CollSafetyClear";
 ELSE
   MoveJ ToPoint,Speed,fine,Tool\WObj?Wobj;
   CollSafetyClear;
 ENDIF
 !
BACKWARD
 !
 MoveJ ToPoint,Speed,fine,Tool\WObj?Wobj;
 !
 CheckValue Coll, 1, 62, 0, "Coll Number";
 IF Present(Coll_B) CheckValue Coll_B, 1, 62, 0, "Coll Number";
 IF Present(Coll_C) CheckValue Coll_C, 1, 62, 0, "Coll Number";
 IF Present(Coll_D) CheckValue Coll_D, 1, 62, 0, "Coll Number";
 IF Present(Coll_E) CheckValue Coll_E, 1, 62, 0, "Coll Number";
 !
 CollSafetyRequest Coll,"";
 IF Present(Coll_B) CollSafetyRequest Coll_B,"";
 IF Present(Coll_C) CollSafetyRequest Coll_C,"";
 IF Present(Coll_D) CollSafetyRequest Coll_D,"";
 IF Present(Coll_E) CollSafetyRequest Coll_E,"";
 !
 ERROR
 !** Error Handler**
 SkipWarn;
 IF ERRNO = ERR_WAIT_MAXTIME TRYNEXT;
ENDPROC !(MoveJ_CollClr)

!*******************************************************************************

PROC MoveL_CollClr( num Coll \num Coll_B  \num Coll_C  \num Coll_D  \num Coll_E, robtarget ToPoint, speeddata Speed, zonedata Zone, PERS tooldata Tool \PERS wobjdata Wobj)
 !*************************************************************
 !*               Procedure MoveLCollClr                      *
 !*     Modified MoveL with Triggering of CollSafety Clear    *
 !*************************************************************
 VAR btnres br_UiAnswer;
 VAR bool b_TimeOut;
 VAR errnum errno1;
 !
 CheckValue Coll, 1, 62, 0, "Coll Number";
 IF Present(Coll_B) CheckValue Coll_B, 1, 62, 0, "Coll Number";
 IF Present(Coll_C) CheckValue Coll_C, 1, 62, 0, "Coll Number";
 IF Present(Coll_D) CheckValue Coll_D, 1, 62, 0, "Coll Number";
 IF Present(Coll_E) CheckValue Coll_E, 1, 62, 0, "Coll Number";
 !
 !Warten bis vorherige Bearbeitung erledigt
 !
 WaitUntil b_CollClearAct=FALSE\MaxTime:=3\TimeFlag:=b_TimeOut;
 !*************************************************************
 !*   Waiting for acknowledge that the Collsion was released  *
 !*************************************************************
 IF b_CollClearAct=TRUE THEN
   IF OpMode()= OP_MAN_PROG THEN
	st_UiHeader:=["Com, CollZoneClearError","Com, CollZoneClearError","???"];
	st_UiMsgLine1:=["Warning","Achtung","???"];
	st_UiMsgLine2:=["","","???"];
	st_UiMsgLine3:=["The clear collision zone routine was interrupted!","Die Funktion loesche Kollisionsschutz wurde abgebrochen","???"];
	st_UiMsgLine4:=["Please confirm in Manual Mode! ","Bestaetige in Handbetrieb","???"];
	UIMsgBox\Header:=st_UiHeader{n_Sp},st_UiMsgLine1{n_Sp}\MsgLine2:=st_UiMsgLine2{n_Sp}
  		\MsgLine3:=st_UiMsgLine3{n_Sp}\MsgLine4:=st_UiMsgLine4{n_Sp}
	 	\Buttons:=btnOK\Icon:=iconError;
     	b_CollClearAct:=FALSE;
   ELSE
	WHILE b_CollClearAct=TRUE DO
	st_UiHeader:=["Com, CollZoneClearError","Com, CollZoneClearError","???"];
	st_UiMsgLine2:=["MoveLCollClr: Wait b_CollClearAct=FALSE","MoveLCollClr: Warte auf b_CollClearAct=FALSE","???"];
	st_UiMsgLine3:=["The clear function has not been finished yet","Das Freigeben der Zone ist noch nicht abgeschlossen!","???"];
	UIMsgBox\Header:=st_UiHeader{n_Sp},""\MsgLine2:=st_UiMsgLine2{n_Sp}\MsgLine3:=st_UiMsgLine3{n_Sp}
		\Buttons:=btnNone\Icon:=iconWarning\MaxTime:=1\BreakFlag:=errno1;
     ENDWHILE
   ENDIF
 ENDIF
 !
 !In bearbeitung
 b_CollClearAct:=TRUE;
 !
 !Init Zonen / Init zone
 !
 FOR i FROM 1 TO 5 DO
   n_Coll{i}:=0;
 ENDFOR
 !
 !Einlesen der Zonen / Reading the Zone
 !
 n_CollClZ:=1;
 n_Coll{1}:=Coll;
 !
 IF Present(Coll_B) THEN
   Incr n_CollClZ;
   n_Coll{2}:=Coll_B;
 ENDIF
 !
 IF Present(Coll_C) THEN
   Incr n_CollClZ;
   IF n_Coll{2}=0 THEN
     n_Coll{2}:=Coll_C;
   ELSE
     n_Coll{3}:=Coll_C;
   ENDIF
 ENDIF
 !
 IF Present(Coll_D) THEN
   Incr n_CollClZ;
   IF n_Coll{2}=0 THEN
     n_Coll{2}:=Coll_D;
   ELSE
     IF n_Coll{3}=0 THEN
       n_Coll{3}:=Coll_D;
     ELSE
       n_Coll{4}:=Coll_D;
     ENDIF
   ENDIF
 ENDIF
 !
 IF Present(Coll_E) THEN
   Incr n_CollClZ;
   IF n_Coll{2}=0 THEN
     n_Coll{2}:=Coll_E;
   ELSE
     IF n_Coll{3}=0 THEN
       n_Coll{3}:=Coll_E;
     ELSE
       IF n_Coll{4}=0 THEN
         n_Coll{4}:=Coll_E;
       ELSE
         n_Coll{5}:=Coll_E;
       ENDIF
     ENDIF
   ENDIF
 ENDIF
 !
 !Wenn nicht besetzt / When not occupied
 !
 FOR i FROM 1 TO n_CollClZ DO
   IF OpMode()= OP_AUTO THEN
     WHILE b_CollZoneOccupied{n_Coll{i}}=FALSE DO
		st_MsgBoxHeader:=["Com, MoveLCollClr","Com, Kollisionsschutzfreigabe","Com,???"];
   	st_Dummy:=["CollZone= "+NumToStr(n_Coll{i},0),"CollZone= "+NumToStr(n_Coll{i},0),"???"];
   	st_Dummy2:=["is not already requested!","war nicht angefragt!","???"];
   	st_MsgBoxbutton4:=["Ok","Ok","???"];
   	st_MsgBoxbutton5:=["","","???"];
   	n_MsgBoxApplError:=0;
   	n_MsgBoxPLC_Error:=51;
   	st_MsgBoxElogLine4:="ComBase/MoveLCollClr";
   	MsgBox\diBreakSignal:=SYS_di_ErrReset\Line1:=st_Dummy{n_Sp}\Line2:=st_Dummy2{n_Sp}\ErrorToPLC;
	!
     ENDWHILE
   ELSE
     IF b_CollZoneOccupied{n_Coll{i}}=FALSE THEN
       st_UiHeader:=["Com, MoveLCollClr","Com, Kollisionsschutzfreigabe","???"];
			st_UiMsgLine1:=["Clear Error","Freigabefehler!","???"];
			st_UiMsgLine2:=["is not already requested!","Bereich war nicht angefragt!","???"];
			st_UiMsgLine3:=["Please check the collisions zones already","ueberpruefe den Status der Kollisionszone","???"];
			st_UiMsgLine4:=["requested and confirm their status. ","Bestaetige den Zustand !","???"];
			UIMsgBox\Header:=st_UiHeader{n_Sp},st_UiMsgLine1{n_Sp}\MsgLine2:=st_UiMsgLine2{n_Sp}
  			\MsgLine3:=st_UiMsgLine3{n_Sp}\MsgLine4:=st_UiMsgLine4{n_Sp}\Buttons:=btnOK\Icon:=iconWarning;
     ENDIF
   ENDIF
 ENDFOR
 !
 IF RunMode() = RUN_CONT_CYCLE THEN
   MoveLSync ToPoint,Speed, Zone,Tool\WObj?Wobj, "CollSafetyClear";
 ELSE
   MoveL ToPoint,Speed,fine,Tool\WObj?Wobj;
   CollSafetyClear;
 ENDIF
 !
 BACKWARD
 !
 MoveL ToPoint,Speed,fine,Tool\WObj?Wobj;
 !
 CheckValue Coll, 1, 62, 0, "Coll Number";
 IF Present(Coll_B) CheckValue Coll_B, 1, 62, 0, "Coll Number";
 IF Present(Coll_C) CheckValue Coll_C, 1, 62, 0, "Coll Number";
 IF Present(Coll_D) CheckValue Coll_D, 1, 62, 0, "Coll Number";
 IF Present(Coll_E) CheckValue Coll_E, 1, 62, 0, "Coll Number";
 !
 CollSafetyRequest Coll,"";
 IF Present(Coll_B) CollSafetyRequest Coll_B,"";
 IF Present(Coll_C) CollSafetyRequest Coll_C,"";
 IF Present(Coll_D) CollSafetyRequest Coll_D,"";
 IF Present(Coll_E) CollSafetyRequest Coll_E,"";
 !
 ERROR
 !** Error Handler**
 SkipWarn;
 IF ERRNO = ERR_WAIT_MAXTIME TRYNEXT;
ENDPROC !(MoveL_CollClr)

!*******************************************************************************

